(* IEC 61131-3 sources: plc_projects/St_Codes, 9 files *)

(* ---- GVL.st ---- *)
(* ==========================================
   POU: GVL
   ========================================== *)

=== DECLARATION ===
{attribute 'qualified_only'}
VAR_GLOBAL
    Recipe_Weights AT %MD100 : ARRAY[1..20] OF REAL;
	Auto_Bin_Material_Mapping AT %MW50: ARRAY[1..6] OF INT;
	Semi_Auto_Bin_Material_Mapping AT %MW60: ARRAY[1..10] OF INT;
	Auto_Coarse_To_Fine_speed AT %MD120: ARRAY[1..6] OF REAL := [1.0,1.0,1.0,1.0,1.0,1.0];
	Semi_Auto_Coarse_To_Fine_speed AT %MD130: ARRAY[1..10] OF REAL := [1.0,1.0,1.0,1.0,1.0,1.0,1.0,1.0,1.0,1.0];
	Auto_Bin_Tolerance AT %MD150: ARRAY[1..6] OF REAL;
	Semi_Auto_Bin_Tolerance AT %MD160: ARRAY[1..10] OF REAL;
	Start_Button AT %MX2.0: BOOL;
	E_Stop_Active AT %MX2.1: BOOL;
	Reset AT %MX2.3: BOOL;
	Next_Cycle_Start AT %MX2.4: BOOL;               // Command pulse/signal to start next batch cycle after hoppers are emptied
	Auto_Active_Mat AT %MW70: INT;
	Auto_Active_Bin AT %MW71: INT;
	Semi_Auto_Active_Mat AT %MW72: INT;
	Semi_Auto_Active_Bin AT %MW73: INT;
	Target_Batch_Cycles AT %MW74: INT := 1;
	Current_Batch_Cycle AT %MW75: INT;
	Completed_Batch_Cycles AT %MW79: INT;
	Error_Code AT %MW76: INT;
	Run AT %MX2.5 : BOOL;
	load_cell_auto AT %MD174 : REAL;
	load_cell_semi_auto AT %MD175 : REAL;
	Auto_Initial_Tolerance AT %MD176 : REAL := 5.0;
	Semi_Auto_Initial_Tolerance AT %MD178 : REAL := 5.0;
	Empty_Weight_Limit AT %MD186 : REAL := 5.0;     // Maximum scale weight limit (kg) to qualify scale as empty before starting next cycle
	Auto_Total_Target_Weight AT %MD180 : REAL;
	Semi_Auto_Total_Target_Weight AT %MD184 : REAL;
	Auto_Material_Count AT %MW77 : INT;
	Semi_Auto_Material_Count AT %MW78 : INT;
	Auto_Current_Step AT %MW80 : INT;
	Semi_Auto_Current_Step AT %MW81 : INT;
	Auto_Active_Target_Weight AT %MD220 : REAL;
	Semi_Auto_Active_Target_Weight AT %MD224 : REAL;
	Auto_Active_Live_Weight AT %MD228 : REAL;
	Semi_Auto_Active_Live_Weight AT %MD232 : REAL;
	Auto_Excess_Allowed AT %MX2.6 : BOOL;
	Semi_Auto_Excess_Allowed AT %MX2.9 : BOOL;
	Auto_Excess_Alarm AT %MX2.7 : BOOL;
	Semi_Auto_Excess_Alarm AT %MX2.8 : BOOL;
	Auto_Inter_Bin_Delay AT %MD190 : TIME;
	Semi_Auto_Inter_Bin_Delay AT %MD194 : TIME;
	Auto_Sequence_Complete AT %MX3.0 : BOOL;
	Semi_Auto_Sequence_Complete AT %MX3.1 : BOOL;
	All_Cycles_Complete AT %MX3.2 : BOOL;           // Master flag: TRUE when all target batch cycles have completed
	Auto_Status_Message : STRING(80);
	Semi_Auto_Status_Message : STRING(80);

	(* 8 Process Output and Weight Arrays *)
	Auto_Bin : ARRAY[1..6] OF BOOL;
	auto_bin_cutoff : ARRAY[1..6] OF BOOL;
	auto_bin_motor : ARRAY[1..6] OF BOOL;
	Semi_Auto_Bin : ARRAY[1..10] OF BOOL;
	semi_auto_bin_cutoff : ARRAY[1..10] OF BOOL;
	semi_auto_bin_motor : ARRAY[1..10] OF BOOL;
	Auto_Weights : ARRAY[1..6] OF REAL;
	Semi_Auto_Weights : ARRAY[1..10] OF REAL;
END_VAR

(* ---- Auto_Batching_V13.st ---- *)
FUNCTION_BLOCK Auto_Batching_V13
VAR_INPUT
    Start_Button : BOOL;      // Signal to start/resume the batching sequence
    E_Stop_Active : BOOL;     // Emergency Stop (Pause/Hold signal)
    Reset : BOOL;             // Hard reset sequence trigger
    Auto_Bin_Material_Mapping : ARRAY[1..6] OF INT; // Material index mapping for 6 bins
    Auto_Coarse_To_Fine_speed : ARRAY[1..6] OF REAL; // Cutoff weight thresholds (kg)
    Auto_Bin_Tolerance : ARRAY[1..6] OF REAL; // Tolerance weight offset values (kg)
    Inter_Bin_Delay : TIME;   // Global inter-bin delay time
    Excess_Allowed : BOOL;    // Global toggle: TRUE = skip excess check, FALSE = trigger alarm & hold
END_VAR
VAR_IN_OUT
    load_cell_value : REAL;   // Weight value read/written from load cell
END_VAR
VAR_OUTPUT
    Auto_Bin : ARRAY[1..6] OF BOOL; // Coarse feed valve outputs
    auto_bin_cutoff : ARRAY[1..6] OF BOOL; // Fine feed cutoff trigger indicators
    auto_bin_motor : ARRAY[1..6] OF BOOL; // Main conveyor motor outputs
    Actual_Weights : ARRAY[1..6] OF REAL; // Actual weight poured per silo
    Sequence_Complete : BOOL;  // Batch complete flag
    Active_Material_ID : INT;  // Currently active ingredient ID
    Active_Bin_ID : INT;       // Currently active physical Bin ID (1..6)
    Active_Target_Weight : REAL; // Recipe target weight of active bin
    Active_Live_Weight : REAL; // Live tared weight poured from active bin
    Excess_Alarm : BOOL;       // Excess weight alarm output
    Error_Code : INT;          // Active error code
    Status_Message : STRING;   // Diagnostic text message
END_VAR
VAR
    Step : INT;                // State machine index (0: Idle, 1..6: Pour, 7: Settling, 8: Complete)
    bin_last_weight : REAL;   // Baseline weight snapshot before starting current bin
    actual_bin : REAL;        // Current weight added from active bin
    target_weight : REAL;     // Target recipe weight
    cutoff_trigger_weight : REAL; // Calculated cutoff trigger threshold (Target - Cutoff)
    min_tol_weight : REAL;    // Minimum allowable tolerance (Target - Tol)
    max_tol_weight : REAL;    // Maximum allowable tolerance (Target + Tol)
    Paused_By_EStop : BOOL;    // Pause status latch
    Effective_Delay : TIME;   // Resolved delay time (defaults to T#2S if T#0S configured)

    Mat_Idx : INT;
    i : INT;                  // General loop index

    (* TIMERS FOR TRANSITIONS & DELAYS *)
    Transition_Timer : TON;
    Completion_Timer : TON;

    (* SELF-CONTAINED SIMULATION VARIABLES *)
    Simulation_Mode : BOOL;    // Simulation disabled for physical PLC use
    Sim_Rate : REAL;
    Sim_Timer : TON;
    Start_Sim_Weight : REAL;
    Discharge_Active : BOOL;
END_VAR

(* Auto Batching FB V13 with Real-Time Instant Excess Verification & Clean Multi-Cycle Reset *)

Effective_Delay := Inter_Bin_Delay;
IF Effective_Delay = T#0S THEN
    Effective_Delay := T#2S;
END_IF;

(* 1. HARD RESET INTERLOCK *)
IF Reset THEN
    FOR i := 1 TO 6 DO
        Auto_Bin[i] := FALSE;
        auto_bin_cutoff[i] := FALSE;
        auto_bin_motor[i] := FALSE;
        Actual_Weights[i] := 0.0;
    END_FOR;
    Sequence_Complete := FALSE;
    Active_Material_ID := 0;
    Active_Bin_ID := 0;
    Active_Target_Weight := 0.0;
    Active_Live_Weight := 0.0;
    Excess_Alarm := FALSE;
    Error_Code := 0;
    Status_Message := '';
    Paused_By_EStop := FALSE;
    Step := 0;

    bin_last_weight := 0.0;
    Start_Sim_Weight := 0.0;

    Transition_Timer(IN := FALSE);
    Completion_Timer(IN := FALSE);
    Sim_Timer(IN := FALSE);
    RETURN;
END_IF;

(* 2. E-STOP PAUSE / HOLD LOGIC *)
IF E_Stop_Active THEN
    Paused_By_EStop := TRUE;
END_IF;

IF Paused_By_EStop THEN
    FOR i := 1 TO 6 DO
        Auto_Bin[i] := FALSE;
        auto_bin_cutoff[i] := FALSE;
        auto_bin_motor[i] := FALSE;
    END_FOR;

    IF E_Stop_Active THEN
        Status_Message := 'Auto Paused: Emergency Stop Active!';
    ELSE
        Status_Message := 'Auto Paused: Press Start to Resume';
        IF Start_Button THEN
            Paused_By_EStop := FALSE;
        END_IF;
    END_IF;

    Sim_Timer(IN := FALSE);
    Transition_Timer(IN := FALSE);
    Completion_Timer(IN := FALSE);
    RETURN;
END_IF;

(* 3. SIMULATION WEIGHT MANAGEMENT (WHEN ENABLED) *)
IF Simulation_Mode THEN
    IF Step = 0 AND NOT Start_Button AND NOT Sequence_Complete THEN
        load_cell_value := 0.0;
        bin_last_weight := 0.0;
        Start_Sim_Weight := 0.0;
        Sim_Timer(IN := FALSE);
    END_IF;

    Discharge_Active := FALSE;
    IF Step >= 1 AND Step <= 6 THEN
        Discharge_Active := auto_bin_motor[Step];
    END_IF;

    IF Discharge_Active THEN
        Sim_Timer(IN := TRUE, PT := T#1000S);
        load_cell_value := Start_Sim_Weight + (TIME_TO_REAL(Sim_Timer.ET) / 1000.0) * Sim_Rate;
    ELSE
        Sim_Timer(IN := FALSE);
        Start_Sim_Weight := load_cell_value;
    END_IF;
END_IF;

(* 4. RECIPE SEQUENCE START & CYCLIC RESET *)
IF Step = 0 AND Start_Button THEN
    Step := 1;
    bin_last_weight := load_cell_value; (* Snapshot relative tare at whatever weight scale is *)
    Sequence_Complete := FALSE;
    Excess_Alarm := FALSE;
    Error_Code := 0;
    Status_Message := 'Auto Pour Started';
    Active_Target_Weight := 0.0;
    Active_Live_Weight := 0.0;
    FOR i := 1 TO 6 DO
        Actual_Weights[i] := 0.0;
        Auto_Bin[i] := FALSE;
        auto_bin_cutoff[i] := FALSE;
        auto_bin_motor[i] := FALSE;
    END_FOR;
END_IF;

(* 5. SEQUENCE CONTROL STATE MACHINE *)
CASE Step OF
    0:
        Active_Material_ID := 0;
        Active_Bin_ID := 0;
        Active_Target_Weight := 0.0;
        Active_Live_Weight := 0.0;
        Excess_Alarm := FALSE;
        Sequence_Complete := FALSE;
        FOR i := 1 TO 6 DO
            Auto_Bin[i] := FALSE;
            auto_bin_cutoff[i] := FALSE;
            auto_bin_motor[i] := FALSE;
        END_FOR;
        IF Error_Code = 0 THEN Status_Message := 'Auto Idle'; END_IF;

    1..6: (* DISCHARGE SILOS 1 TO 6 *)
        Mat_Idx := Auto_Bin_Material_Mapping[Step];

        (* Skip this step instantly if material mapping is 0 OR target weight is 0.0 kg *)
        IF Mat_Idx = 0 OR (Mat_Idx <= 20 AND GVL.Recipe_Weights[Mat_Idx] = 0.0) THEN
            IF Step = 6 THEN
                Step := 7; (* Transition directly to final settling delay *)
            ELSE
                Step := Step + 1;
            END_IF;
        ELSE
            target_weight := GVL.Recipe_Weights[Mat_Idx];
            cutoff_trigger_weight := target_weight - Auto_Coarse_To_Fine_speed[Step];
            min_tol_weight := target_weight - Auto_Bin_Tolerance[Step];
            max_tol_weight := target_weight + Auto_Bin_Tolerance[Step];

            Active_Target_Weight := target_weight;
            actual_bin := load_cell_value - bin_last_weight;
            Actual_Weights[Step] := actual_bin;
            Active_Live_Weight := actual_bin; (* Live tared weight of active bin *)

            Active_Material_ID := Mat_Idx;
            Active_Bin_ID := Step;

            (* Scale Overload Protection *)
            IF load_cell_value > 500.0 THEN
                Error_Code := 21;
                Status_Message := 'Error 21: Scale Overloaded!';
                Sequence_Complete := TRUE;
                Paused_By_EStop := TRUE;
            END_IF;

            (* Real-Time Feed & Instant Excess Alarm *)
            IF actual_bin < cutoff_trigger_weight THEN
                (* Coarse Feed *)
                Auto_Bin[Step] := TRUE;
                auto_bin_cutoff[Step] := FALSE;
                auto_bin_motor[Step] := TRUE;
                Excess_Alarm := FALSE;
                Status_Message := 'Auto Pouring (Coarse Feed)';

            ELSIF actual_bin < min_tol_weight THEN
                (* Fine Feed *)
                Auto_Bin[Step] := FALSE;
                auto_bin_cutoff[Step] := TRUE;
                auto_bin_motor[Step] := TRUE;
                Excess_Alarm := FALSE;
                Status_Message := 'Auto Pouring (Fine Feed)';

            ELSIF actual_bin > max_tol_weight THEN
                (* Excess Weight -> Instant Alarm, No Delay! *)
                Auto_Bin[Step] := FALSE;
                auto_bin_cutoff[Step] := FALSE;
                auto_bin_motor[Step] := FALSE;

                IF Excess_Allowed THEN
                    Excess_Alarm := FALSE;
                    Status_Message := 'Excess Weight Allowed: Advancing';
                    bin_last_weight := load_cell_value;
                    Active_Target_Weight := 0.0;
                    Active_Live_Weight := 0.0;
                    IF Step = 6 THEN
                        Step := 7;
                    ELSE
                        Step := Step + 1;
                    END_IF;
                ELSE
                    Excess_Alarm := TRUE; (* Immediate Trigger! *)
                    Status_Message := 'Excess Alarm: Weight above max tolerance! Reduce weight.';
                END_IF;

            ELSE
                (* In Tolerance Window [Min_Tol .. Max_Tol] *)
                Auto_Bin[Step] := FALSE;
                auto_bin_cutoff[Step] := FALSE;
                auto_bin_motor[Step] := FALSE;
                Excess_Alarm := FALSE;
                bin_last_weight := load_cell_value;
                Active_Target_Weight := 0.0;
                Active_Live_Weight := 0.0;

                IF Step = 6 THEN
                    Step := 7;
                ELSE
                    Step := Step + 1;
                END_IF;
            END_IF;
        END_IF;

    7: (* POST-SEQUENCE FINAL SETTLING DELAY *)
        Active_Material_ID := 0;
        Active_Bin_ID := 0;
        Active_Target_Weight := 0.0;
        Active_Live_Weight := 0.0;
        Excess_Alarm := FALSE;
        Status_Message := 'Final Settling Delay';
        Completion_Timer(IN := TRUE, PT := Effective_Delay);
        IF Completion_Timer.Q THEN
            Completion_Timer(IN := FALSE);
            Step := 8;
        END_IF;

    8: (* COMPLETE *)
        Active_Material_ID := 0;
        Active_Bin_ID := 0;
        Active_Target_Weight := 0.0;
        Active_Live_Weight := 0.0;
        Excess_Alarm := FALSE;
        Status_Message := 'Sequence Completed';
        Sequence_Complete := TRUE;

        IF NOT Start_Button THEN
            Step := 0;
            Sequence_Complete := FALSE;
            FOR i := 1 TO 6 DO
                Actual_Weights[i] := 0.0;
            END_FOR;
        END_IF;
END_CASE;

(* ---- Auto_Batching_V14.st ---- *)
FUNCTION_BLOCK Auto_Batching_V14
VAR_INPUT
    Start_Button : BOOL;                            // Command pulse/signal to start or resume the auto batching sequence
    E_Stop_Active : BOOL;                           // Emergency Stop circuit status (NC contact: TRUE = Healthy/Run permitted, FALSE = E-Stop tripped)
    Reset : BOOL;                                   // System reset pulse (clears active steps, outputs, alarms, and error flags)
    Auto_Bin_Material_Mapping : ARRAY[1..6] OF INT; // Array mapping physical Silos 1..6 to Recipe Material IDs (1..20, 0 = Silo skipped)
    Auto_Coarse_To_Fine_Speed : ARRAY[1..6] OF REAL;// Weight offset threshold (kg) before target to transition from Coarse to Fine feeding
    Auto_Bin_Tolerance : ARRAY[1..6] OF REAL;       // Allowable weight tolerance window (±kg) around target weight for each silo
    Inter_Bin_Delay : TIME;                         // Settling delay duration after completing a bin before advancing to the next
    Excess_Allowed : BOOL;                          // Overfill handling policy: TRUE = proceed if target is exceeded, FALSE = raise alarm and halt
    load_cell_value : REAL;                         // Live gross weight input reading from the Auto scale load cell (kg)
    Target_Batch_Cycles : INT;                      // Target number of batch cycle repetitions configured from HMI (defaults to 1)
    Next_Cycle_Start : BOOL;                        // Command pulse/signal to start next batch cycle after hoppers are emptied
    Empty_Weight_Limit : REAL;                      // Maximum scale weight limit (kg) for scales to qualify as empty before starting next cycle
END_VAR
VAR_OUTPUT
    Auto_Bin : ARRAY[1..6] OF BOOL;                 // Coarse feeding valve / gate actuation command outputs for Silos 1..6
    auto_bin_cutoff : ARRAY[1..6] OF BOOL;          // Fine feeding valve / vibrator cutoff actuation command outputs for Silos 1..6
    auto_bin_motor : ARRAY[1..6] OF BOOL;           // Feeder / screw conveyor motor run commands for Silos 1..6
    Actual_Weights : ARRAY[1..6] OF REAL;           // Net material weight (kg) successfully dosed for each silo in the current cycle
    Sequence_Complete : BOOL;                       // Handshake flag: TRUE when all mapped Auto silos have completed dosing and settling
    Active_Material_ID : INT;                       // Recipe Material ID currently being dosed (1..20, 0 when idle/complete)
    Active_Bin_ID : INT;                            // Physical Silo index currently being dosed (1..6, 0 when idle/complete)
    Active_Target_Weight : REAL;                    // Target weight setpoint (kg) of the ingredient currently being dosed
    Active_Live_Weight : REAL;                      // Live net/tared weight (kg) accumulated into the scale for the active silo
    Current_Step : INT;                             // Real-time sequence step:
                                                    //   0  = Idle / Waiting for Start
                                                    //   1..6 = Dosing Silos 1..6 (feeding coarse/fine)
                                                    //   7  = Settling delay in progress
                                                    //   8  = Sequence complete
    Cycle_Manager_State : INT;                      // Master supervisory cycle manager state:
                                                    //   0  = System Idle / Stopped
                                                    //   1  = Running active batch cycle
                                                    //   4  = All target batch cycles completed successfully
                                                    //   5  = Paused between cycles (Cycle Hold active)
    Excess_Alarm : BOOL;                            // Overfill alarm: TRUE when dosed weight exceeds target + tolerance (with Excess_Allowed=FALSE)
    Error_Code : INT;                               // Fault diagnostic code:
                                                    //   0  = No Error / System Healthy
                                                    //   1  = Duplicate Material ID mapped across Auto and Semi-Auto
                                                    //   2  = Material index out of range (must be 1..20)
                                                    //   3  = Recipe weight is less than (Coarse_To_Fine_Speed + Tolerance)
                                                    //   4  = Initial scale tare error (scale not empty before start)
                                                    //   21 = Scale overload protection triggered (> 500 kg)
    Auto_Current_Batch_Cycle : INT;                     // Active batch cycle number currently processing (1..Target_Batch_Cycles)
    Auto_Completed_Batch_Cycles : INT;                  // Total number of batch cycle loops completed successfully
    Auto_All_Cycles_Complete : BOOL;                    // Master flag: TRUE when all Target_Batch_Cycles have finished
    Status_Message : STRING(80);                    // Real-time human-readable process status and diagnostic text message
END_VAR
VAR
    bin_last_weight : REAL;
    actual_bin : REAL;
    target_weight : REAL;
    cutoff_trigger_weight : REAL;
    min_tol_weight : REAL;
    max_tol_weight : REAL;
    Paused_By_EStop : BOOL;
    Effective_Delay : TIME;
    Mat_Idx : INT;
    i : INT;
    j : INT;
    Transition_Timer : TON;
    Completion_Timer : TON;
    Simulation_Mode : BOOL;
    Sim_Rate : REAL;
    Sim_Timer : TON;
    Start_Sim_Weight : REAL;
    Discharge_Active : BOOL;

    (* Master Cycle Manager & Supervisory states *)
    Internal_FB_Start : BOOL;
    Duplicate_Found : BOOL;
    Invalid_Material_Range : BOOL;
    Weight_Limit_Error : BOOL;
    eff_empty_limit : REAL;
    Next_Cycle_Last : BOOL;
    Next_Cycle_Rising : BOOL;
END_VAR

(* Auto Batching FB V14 with Full Diagnostics, Step Tracking, and Precise Status Reporting *)

Effective_Delay := Inter_Bin_Delay;
IF Effective_Delay = T#0S THEN
    Effective_Delay := T#2S;
END_IF;

(* Detect rising edge on Next_Cycle_Start trigger *)
Next_Cycle_Rising := (Next_Cycle_Start OR GVL.Next_Cycle_Start) AND NOT Next_Cycle_Last;
Next_Cycle_Last := (Next_Cycle_Start OR GVL.Next_Cycle_Start);

(* 1. RECIPE TOTALS & SUPERVISORY CONFIGURATION CHECKS *)
Duplicate_Found := FALSE;
Invalid_Material_Range := FALSE;
Weight_Limit_Error := FALSE;

GVL.Auto_Total_Target_Weight := 0.0;
GVL.Auto_Material_Count := 0;
FOR i := 1 TO 6 DO
    IF Auto_Bin_Material_Mapping[i] < 0 OR Auto_Bin_Material_Mapping[i] > 20 THEN
        Invalid_Material_Range := TRUE;
    END_IF;
    IF Auto_Bin_Material_Mapping[i] <> 0 AND Auto_Bin_Material_Mapping[i] <= 20 THEN
        FOR j := 1 TO 10 DO
            IF Auto_Bin_Material_Mapping[i] = GVL.Semi_Auto_Bin_Material_Mapping[j] THEN
                Duplicate_Found := TRUE;
            END_IF;
        END_FOR;
    END_IF;
    IF Auto_Bin_Material_Mapping[i] > 0 AND Auto_Bin_Material_Mapping[i] <= 20 THEN
        IF GVL.Recipe_Weights[Auto_Bin_Material_Mapping[i]] > 0.0 THEN
            GVL.Auto_Total_Target_Weight := GVL.Auto_Total_Target_Weight + GVL.Recipe_Weights[Auto_Bin_Material_Mapping[i]];
            GVL.Auto_Material_Count := GVL.Auto_Material_Count + 1;
            IF GVL.Recipe_Weights[Auto_Bin_Material_Mapping[i]] < (Auto_Coarse_To_Fine_Speed[i] + Auto_Bin_Tolerance[i]) THEN
                Weight_Limit_Error := TRUE;
            END_IF;
        END_IF;
    END_IF;
END_FOR;

IF Duplicate_Found THEN
    GVL.Error_Code := 1;
    Error_Code := 1;
    Status_Message := 'Error 1: Duplicate Material ID mapped in Auto and Semi-Auto!';
ELSIF Invalid_Material_Range THEN
    GVL.Error_Code := 2;
    Error_Code := 2;
    Status_Message := 'Error 2: Material Index configuration out of range (1..20)!';
ELSIF Weight_Limit_Error THEN
    GVL.Error_Code := 3;
    Error_Code := 3;
    Status_Message := 'Error 3: Recipe weight is less than Coarse_To_Fine_Speed + Tolerance!';
ELSE
    IF GVL.Error_Code <= 3 THEN
        GVL.Error_Code := 0;
        Error_Code := 0;
    END_IF;
END_IF;

(* 2. HARD RESET INTERLOCK *)
IF Reset OR GVL.Reset THEN
    FOR i := 1 TO 6 DO
        Auto_Bin[i] := FALSE;
        auto_bin_cutoff[i] := FALSE;
        auto_bin_motor[i] := FALSE;
        Actual_Weights[i] := 0.0;
        GVL.Auto_Bin[i] := FALSE;
        GVL.auto_bin_cutoff[i] := FALSE;
        GVL.auto_bin_motor[i] := FALSE;
        GVL.Auto_Weights[i] := 0.0;
    END_FOR;

    (* Reset Recipe & Active Target Setpoints *)
    FOR i := 1 TO 20 DO
        GVL.Recipe_Weights[i] := 0.0;
    END_FOR;
    GVL.Auto_Total_Target_Weight := 0.0;
    GVL.Semi_Auto_Total_Target_Weight := 0.0;
    GVL.Auto_Material_Count := 0;
    GVL.Semi_Auto_Material_Count := 0;

    Sequence_Complete := FALSE;
    GVL.Auto_Sequence_Complete := FALSE;
    GVL.Semi_Auto_Sequence_Complete := FALSE;
    Active_Material_ID := 0;
    Active_Bin_ID := 0;
    Active_Target_Weight := 0.0;
    Active_Live_Weight := 0.0;
    GVL.Auto_Active_Target_Weight := 0.0;
    GVL.Auto_Active_Live_Weight := 0.0;
    Excess_Alarm := FALSE;
    Error_Code := 0;
    GVL.Error_Code := 0;
    GVL.Current_Batch_Cycle := 0;
    GVL.Completed_Batch_Cycles := 0;
    GVL.All_Cycles_Complete := FALSE;
    Auto_Completed_Batch_Cycles := 0;
    Auto_Current_Batch_Cycle := 0;
    Auto_All_Cycles_Complete := FALSE;
    GVL.Target_Batch_Cycles := 0;
    GVL.Start_Button := FALSE;
    GVL.Run := FALSE;
    GVL.Next_Cycle_Start := FALSE;
    Next_Cycle_Last := FALSE;
    Next_Cycle_Rising := FALSE;
    GVL.Auto_Active_Mat := 0;
    GVL.Auto_Active_Bin := 0;
    GVL.Auto_Excess_Alarm := FALSE;
    Current_Step := 0;
    Cycle_Manager_State := 0;
    Internal_FB_Start := FALSE;
    bin_last_weight := 0.0;
    Start_Sim_Weight := 0.0;
    Transition_Timer(IN := FALSE);
    Completion_Timer(IN := FALSE);
    Sim_Timer(IN := FALSE);
    Status_Message := 'Auto [Reset]: System Reset Complete - System Idle';
    RETURN;
END_IF;

(* 3. E-STOP PAUSE / HOLD LOGIC (NC Contact: FALSE = Pressed/Tripped, TRUE = Healthy) *)
IF NOT E_Stop_Active OR NOT GVL.E_Stop_Active THEN
    Paused_By_EStop := TRUE;
END_IF;

IF Paused_By_EStop THEN
    FOR i := 1 TO 6 DO
        Auto_Bin[i] := FALSE;
        auto_bin_cutoff[i] := FALSE;
        auto_bin_motor[i] := FALSE;
    END_FOR;
    IF NOT E_Stop_Active OR NOT GVL.E_Stop_Active THEN
        Status_Message := CONCAT('Auto [PAUSED]: E-Stop Active at Step ', INT_TO_STRING(Current_Step));
    ELSE
        Status_Message := CONCAT('Auto [HOLD]: E-Stop Cleared. Press Start to Resume Step ', INT_TO_STRING(Current_Step));
        IF Start_Button OR GVL.Start_Button THEN
            Paused_By_EStop := FALSE;
        END_IF;
    END_IF;
    Sim_Timer(IN := FALSE);
    Transition_Timer(IN := FALSE);
    Completion_Timer(IN := FALSE);
    RETURN;
END_IF;

(* 4. MASTER CYCLE MANAGER STATE MACHINE *)
CASE Cycle_Manager_State OF
    0: (* IDLE *)
        Internal_FB_Start := FALSE;
        GVL.Run := FALSE;
        GVL.Next_Cycle_Start := FALSE;
        GVL.Auto_Sequence_Complete := FALSE;

        IF GVL.Error_Code = 0 AND NOT (Start_Button OR GVL.Start_Button) THEN
            Status_Message := 'Auto [State 0 - Idle]: Ready - Waiting for Start Button';
        END_IF;

        IF Start_Button OR GVL.Start_Button THEN
            (* Use Target_Batch_Cycles from input, or fallback to GVL, or default to 1 *)
            IF Target_Batch_Cycles > 0 THEN
                GVL.Target_Batch_Cycles := Target_Batch_Cycles;
            ELSIF GVL.Target_Batch_Cycles <= 0 THEN
                GVL.Target_Batch_Cycles := 1;
            END_IF;

            IF NOT E_Stop_Active OR NOT GVL.E_Stop_Active THEN
                GVL.Run := FALSE;
                Status_Message := 'Auto [State 0]: Cannot Start - Emergency Stop Contact Open!';
            ELSIF (GVL.Auto_Initial_Tolerance > 0.0 AND (GVL.load_cell_auto > GVL.Auto_Initial_Tolerance OR GVL.load_cell_auto < (-GVL.Auto_Initial_Tolerance))) OR
                  (GVL.Semi_Auto_Initial_Tolerance > 0.0 AND (GVL.load_cell_semi_auto > GVL.Semi_Auto_Initial_Tolerance OR GVL.load_cell_semi_auto < (-GVL.Semi_Auto_Initial_Tolerance))) THEN
                GVL.Run := FALSE;
                GVL.Error_Code := 4;
                Error_Code := 4;
                Status_Message := 'Auto [State 0]: Error 4 - Scale not zeroed (exceeds Initial Tolerance)!';
            ELSE
                GVL.Error_Code := 0;
                Error_Code := 0;
                GVL.Current_Batch_Cycle := 1;
                GVL.Completed_Batch_Cycles := 0;
                GVL.All_Cycles_Complete := FALSE;
                Auto_Completed_Batch_Cycles := 0;
                Auto_Current_Batch_Cycle := 1;
                Auto_All_Cycles_Complete := FALSE;
                GVL.Run := TRUE;
                Internal_FB_Start := TRUE;
                Sequence_Complete := FALSE;
                GVL.Auto_Sequence_Complete := FALSE;
                GVL.Semi_Auto_Sequence_Complete := FALSE;
                Cycle_Manager_State := 1;
                Current_Step := 0;
            END_IF;
        END_IF;

    1: (* RUNNING CYCLE *)
        Internal_FB_Start := TRUE;
        GVL.Run := TRUE;

        (* Interlock: While process is actively running, Next_Cycle_Start MUST be FALSE *)
        GVL.Next_Cycle_Start := FALSE;

        (* Both Auto and Semi-Auto must complete to finish the cycle *)
        IF Sequence_Complete AND GVL.Semi_Auto_Sequence_Complete THEN
            GVL.Completed_Batch_Cycles := GVL.Current_Batch_Cycle;
            Auto_Completed_Batch_Cycles := GVL.Current_Batch_Cycle;
            IF GVL.Current_Batch_Cycle < GVL.Target_Batch_Cycles AND GVL.Error_Code = 0 THEN
                Internal_FB_Start := FALSE;
                Cycle_Manager_State := 5; (* Go to pause/hold to wait for scale empty & Next_Cycle_Start *)
            ELSE
                Cycle_Manager_State := 4; (* All target cycles completed *)
            END_IF;
        END_IF;

    5: (* PAUSED BETWEEN CYCLES - WAITING FOR HOPPERS EMPTIED & NEXT CYCLE START *)
        Internal_FB_Start := FALSE;
        GVL.Run := TRUE;

        (* Determine effective empty weight threshold (defaults to 5.0 kg if <= 0.0) *)
        eff_empty_limit := Empty_Weight_Limit;
        IF eff_empty_limit <= 0.0 THEN
            eff_empty_limit := GVL.Empty_Weight_Limit;
        END_IF;
        IF eff_empty_limit <= 0.0 THEN
            eff_empty_limit := 5.0;
        END_IF;

        Status_Message := CONCAT('Auto [State 5]: Cycle ', CONCAT(INT_TO_STRING(GVL.Current_Batch_Cycle), ' Done. Empty scales < limit and trigger Next_Cycle_Start.'));

        (* Check ONLY on a new trigger pulse (rising edge) of Next_Cycle_Start *)
        IF Next_Cycle_Rising THEN
            (* Check both scales are below the empty weight limit at the moment of trigger *)
            IF (GVL.load_cell_auto < eff_empty_limit) AND (GVL.load_cell_semi_auto < eff_empty_limit) THEN
                (* Scale is empty: momentary reset of command, advance to next cycle *)
                GVL.Next_Cycle_Start := FALSE;
                Next_Cycle_Last := FALSE;
                GVL.Start_Button := TRUE; (* Keep Start_Button TRUE until all cycles are complete! *)
                GVL.Error_Code := 0;
                Error_Code := 0;
                GVL.Current_Batch_Cycle := GVL.Current_Batch_Cycle + 1;
                Auto_Current_Batch_Cycle := GVL.Current_Batch_Cycle;
                Sequence_Complete := FALSE;
                GVL.Auto_Sequence_Complete := FALSE;
                GVL.Semi_Auto_Sequence_Complete := FALSE;
                Current_Step := 0;
                Internal_FB_Start := TRUE;
                Cycle_Manager_State := 1;
                FOR i := 1 TO 6 DO
                    Actual_Weights[i] := 0.0;
                    Auto_Bin[i] := FALSE;
                    auto_bin_cutoff[i] := FALSE;
                    auto_bin_motor[i] := FALSE;
                END_FOR;
            ELSE
                (* Scale not empty yet: reject trigger, reset command, and wait for operator to trigger again *)
                GVL.Next_Cycle_Start := FALSE;
                Next_Cycle_Last := FALSE;
                Status_Message := CONCAT('Auto [State 5]: Scale weight exceeds limit (', CONCAT(REAL_TO_STRING(eff_empty_limit), ' kg)! Empty scales and trigger Next_Cycle_Start again.'));
            END_IF;
        END_IF;

    4: (* ALL CYCLES COMPLETE *)
        Internal_FB_Start := FALSE;
        GVL.Run := FALSE;
        GVL.Start_Button := FALSE;
        Auto_All_Cycles_Complete := TRUE;
        GVL.All_Cycles_Complete := TRUE;
        Sequence_Complete := TRUE;
        GVL.Auto_Sequence_Complete := TRUE;
        GVL.Semi_Auto_Sequence_Complete := TRUE;
        Status_Message := CONCAT('Auto [State 4 - Finished]: All ', CONCAT(INT_TO_STRING(GVL.Target_Batch_Cycles), ' Batch Cycles Completed Successfully'));
        IF Start_Button OR GVL.Start_Button THEN
            (* Reset flags for new batch start *)
            Current_Step := 0;
            Auto_All_Cycles_Complete := FALSE;
            GVL.All_Cycles_Complete := FALSE;
            Sequence_Complete := FALSE;
            GVL.Auto_Sequence_Complete := FALSE;
            GVL.Semi_Auto_Sequence_Complete := FALSE;
            Cycle_Manager_State := 0;
        END_IF;
END_CASE;

(* 5. AUTO SILOS 1..6 POURING SEQUENCE WITH DETAILED STATUS *)
IF Current_Step = 0 AND Internal_FB_Start THEN
    Current_Step := 1;
    bin_last_weight := load_cell_value;
    Sequence_Complete := FALSE;
    GVL.Auto_Sequence_Complete := FALSE;
    Excess_Alarm := FALSE;
    Error_Code := 0;
    FOR i := 1 TO 6 DO
        Actual_Weights[i] := 0.0;
        Auto_Bin[i] := FALSE;
        auto_bin_cutoff[i] := FALSE;
        auto_bin_motor[i] := FALSE;
    END_FOR;
END_IF;

CASE Current_Step OF
    0:
        Active_Material_ID := 0;
        Active_Bin_ID := 0;
        Excess_Alarm := FALSE;
        Sequence_Complete := FALSE;
        FOR i := 1 TO 6 DO
            Auto_Bin[i] := FALSE;
            auto_bin_cutoff[i] := FALSE;
            auto_bin_motor[i] := FALSE;
        END_FOR;
        Active_Target_Weight := GVL.Auto_Active_Target_Weight;
        Active_Live_Weight := 0.0;

    1..6:
        (* Skip any bin where Material Mapping is 0, > 20, or Recipe Weight is 0 *)
        WHILE Current_Step >= 1 AND Current_Step <= 6 DO
            Mat_Idx := Auto_Bin_Material_Mapping[Current_Step];
            IF Mat_Idx = 0 OR Mat_Idx > 20 OR GVL.Recipe_Weights[Mat_Idx] <= 0.0 THEN
                Auto_Bin[Current_Step] := FALSE;
                auto_bin_cutoff[Current_Step] := FALSE;
                auto_bin_motor[Current_Step] := FALSE;
                Actual_Weights[Current_Step] := 0.0;
                IF Current_Step = 6 THEN
                    Current_Step := 7;
                    EXIT;
                ELSE
                    Current_Step := Current_Step + 1;
                END_IF;
            ELSE
                EXIT; (* Valid active recipe silo found *)
            END_IF;
        END_WHILE;

        IF Current_Step = 7 THEN
            Active_Material_ID := 0;
            Active_Bin_ID := 0;
            Active_Target_Weight := 0.0;
            Active_Live_Weight := 0.0;
            GVL.Auto_Active_Target_Weight := 0.0;
            GVL.Auto_Active_Live_Weight := 0.0;
            Status_Message := 'Auto [Step 7]: Settling Delay in progress...';
            Completion_Timer(IN := TRUE, PT := Effective_Delay);
            IF Completion_Timer.Q THEN
                Completion_Timer(IN := FALSE);
                Current_Step := 8;
            END_IF;
        ELSE
            Mat_Idx := Auto_Bin_Material_Mapping[Current_Step];
            target_weight := GVL.Recipe_Weights[Mat_Idx];

            Active_Target_Weight := target_weight;
            GVL.Auto_Active_Target_Weight := target_weight;

            cutoff_trigger_weight := target_weight - Auto_Coarse_To_Fine_Speed[Current_Step];
            min_tol_weight := target_weight - Auto_Bin_Tolerance[Current_Step];
            max_tol_weight := target_weight + Auto_Bin_Tolerance[Current_Step];

            actual_bin := load_cell_value - bin_last_weight;
            IF actual_bin < 0.0 THEN
                actual_bin := 0.0;
            END_IF;
            Actual_Weights[Current_Step] := actual_bin;
            Active_Live_Weight := actual_bin;
            GVL.Auto_Active_Live_Weight := actual_bin;
            Active_Material_ID := Mat_Idx;
            Active_Bin_ID := Current_Step;

            IF load_cell_value > 500.0 THEN
                Error_Code := 21;
                GVL.Error_Code := 21;
                Status_Message := CONCAT('Auto [Step ', CONCAT(INT_TO_STRING(Current_Step), ']: STUCK - Error 21: Scale Overloaded (> 500 kg)!'));
                Sequence_Complete := TRUE;
                GVL.Auto_Sequence_Complete := TRUE;
                Paused_By_EStop := TRUE;
            END_IF;

            IF actual_bin < cutoff_trigger_weight THEN
                Auto_Bin[Current_Step] := TRUE;
                auto_bin_cutoff[Current_Step] := FALSE;
                auto_bin_motor[Current_Step] := TRUE;
                Excess_Alarm := FALSE;
                Status_Message := CONCAT('Auto [Step ', CONCAT(INT_TO_STRING(Current_Step), ']: Coarse Feeding'));
            ELSIF actual_bin < min_tol_weight THEN
                Auto_Bin[Current_Step] := FALSE;
                auto_bin_cutoff[Current_Step] := TRUE;
                auto_bin_motor[Current_Step] := TRUE;
                Excess_Alarm := FALSE;
                Status_Message := CONCAT('Auto [Step ', CONCAT(INT_TO_STRING(Current_Step), ']: Fine Feeding'));
            ELSIF actual_bin > max_tol_weight THEN
                Auto_Bin[Current_Step] := FALSE;
                auto_bin_cutoff[Current_Step] := FALSE;
                auto_bin_motor[Current_Step] := FALSE;
                IF Excess_Allowed THEN
                    Excess_Alarm := FALSE;
                    Status_Message := CONCAT('Auto [Step ', CONCAT(INT_TO_STRING(Current_Step), ']: Excess Allowed - Advancing'));
                    bin_last_weight := load_cell_value;
                    Active_Target_Weight := 0.0;
                    Active_Live_Weight := 0.0;
                    GVL.Auto_Active_Target_Weight := 0.0;
                    GVL.Auto_Active_Live_Weight := 0.0;
                    IF Current_Step = 6 THEN
                        Current_Step := 7;
                    ELSE
                        Current_Step := Current_Step + 1;
                    END_IF;
                ELSE
                    Excess_Alarm := TRUE;
                    Status_Message := CONCAT('Auto [Step ', CONCAT(INT_TO_STRING(Current_Step), ']: STUCK - Excess Weight! Reduce weight or enable Excess Allowed.'));
                END_IF;
            ELSE
                Auto_Bin[Current_Step] := FALSE;
                auto_bin_cutoff[Current_Step] := FALSE;
                auto_bin_motor[Current_Step] := FALSE;
                Excess_Alarm := FALSE;
                bin_last_weight := load_cell_value;
                Active_Target_Weight := 0.0;
                Active_Live_Weight := 0.0;
                GVL.Auto_Active_Target_Weight := 0.0;
                GVL.Auto_Active_Live_Weight := 0.0;
                Status_Message := CONCAT('Auto [Step ', CONCAT(INT_TO_STRING(Current_Step), ']: Target Reached - Advancing'));
                IF Current_Step = 6 THEN
                    Current_Step := 7;
                ELSE
                    Current_Step := Current_Step + 1;
                END_IF;
            END_IF;
        END_IF;

    7:
        Active_Material_ID := 0;
        Active_Bin_ID := 0;
        Excess_Alarm := FALSE;
        Status_Message := 'Auto [Step 7]: Settling Delay in progress...';
        Completion_Timer(IN := TRUE, PT := Effective_Delay);
        IF Completion_Timer.Q THEN
            Completion_Timer(IN := FALSE);
            Current_Step := 8;
        END_IF;

    8:
        Active_Material_ID := 0;
        Active_Bin_ID := 0;
        Excess_Alarm := FALSE;
        Sequence_Complete := TRUE;
        GVL.Auto_Sequence_Complete := TRUE;
        IF NOT GVL.Semi_Auto_Sequence_Complete THEN
            Status_Message := 'Auto [Step 8]: Auto Finished. Waiting for Semi-Auto to complete...';
        ELSE
            Status_Message := 'Auto [Step 8]: Cycle Sequences Complete';
        END_IF;
END_CASE;

(* Synchronize physical output arrays to GVL *)
FOR i := 1 TO 6 DO
    GVL.Auto_Bin[i] := Auto_Bin[i];
    GVL.auto_bin_cutoff[i] := auto_bin_cutoff[i];
    GVL.auto_bin_motor[i] := auto_bin_motor[i];
END_FOR;

(* Synchronize live cycle progress to outputs *)
Auto_Current_Batch_Cycle := GVL.Current_Batch_Cycle;
Auto_Completed_Batch_Cycles := GVL.Completed_Batch_Cycles;
Auto_All_Cycles_Complete := GVL.All_Cycles_Complete;

(* ---- FB_Samyak_Control.st ---- *)
(* ==========================================
   POU: FB_Samyak_Control
   ========================================== *)

=== DECLARATION ===
FUNCTION_BLOCK FB_Samyak_Control
VAR_INPUT
    Com_Slot      : BYTE := 1;     (* PLC COM port *)
    Slave_Dev_ID  : BYTE := 1;     (* Samyak slave ID *)
    iDivisor      : REAL := 10.0;  (* Scale factor: Weight_Scaled = Raw / iDivisor *)
    xTare_In      : BOOL;           (* Logic tare pulse *)
    xManual_Tare  : BOOL;           (* HMI/manual tare pulse *)
END_VAR

VAR_OUTPUT
    xStatus_Done   : BOOL;
    xStatus_Busy   : BOOL;
    xStatus_Error  : BOOL;
    iTotalErrCount : INT := 0;
    xLine_Fault    : BOOL;
    Weight_Raw     : DINT;
    Weight_Scaled  : REAL;
    wError_Code    : WORD; (* Check PLC & SAMYAK BaudRate, DevId, Parity; also check PLC serial port LED blink status and RS485 connection if error repeats *)
END_VAR

VAR
    fbRead         : ModRtuMast;
    fbTare         : ModRtuMast;
    iStep          : INT := 0;
    Samyak_Buffer  : ARRAY[0..17] OF WORD;
    wTareCommand   : WORD := 1;

    rtTareTrig     : R_TRIG;
    rtErrTrig      : R_TRIG;
    tStuckWatchdog : TON;
    tRecoveryTimer : TON;

    xTareReq       : BOOL := FALSE; (* Internal tare request latch *)
END_VAR

=== IMPLEMENTATION ===

(* --- 1) Error Tracking + Auto Recovery --- *)
tStuckWatchdog(IN := (fbRead.Busy OR fbTare.Busy), PT := T#2000MS);

rtErrTrig(CLK := (fbRead.Error OR fbTare.Error));
IF rtErrTrig.Q THEN
    iTotalErrCount := iTotalErrCount + 1;
END_IF

IF fbRead.Done OR fbTare.Done THEN
    iTotalErrCount := 0;
    xLine_Fault := FALSE;
END_IF

IF iTotalErrCount >= 10 THEN
    xLine_Fault := TRUE;
END_IF

tRecoveryTimer(IN := xLine_Fault, PT := T#5S);
IF tRecoveryTimer.Q THEN
    iTotalErrCount := 0;
    xLine_Fault := FALSE;
END_IF

IF tStuckWatchdog.Q THEN
    iStep := 99;
END_IF

(* Capture tare request from either input pulse *)
rtTareTrig(CLK := xTare_In OR xManual_Tare);
IF rtTareTrig.Q THEN
    xTareReq := TRUE;
END_IF

(* --- 2) Modbus State Machine --- *)
CASE iStep OF

    0:  (* Continuous Read *)
        fbTare(Execute := FALSE);

        fbRead(
            Execute := NOT (fbRead.Done OR fbRead.Error OR fbRead.Busy)
                       AND NOT xTareReq
                       AND NOT xLine_Fault,
            COM     := Com_Slot,
            Serv    := Slave_Dev_ID,
            FCT     := 3,
            Addr    := 0,
            Nb      := 2,
            Data    := ADR(Samyak_Buffer[0]),
            Timeout := 400,
            Done    => xStatus_Done,
            Busy    => xStatus_Busy,
            Error   => xStatus_Error,
            ErrorID => wError_Code
        );

        IF xStatus_Done THEN
            Weight_Raw := TO_DINT(SHL(TO_DWORD(Samyak_Buffer[1]), 16) OR TO_DWORD(Samyak_Buffer[0]));
            Weight_Scaled := TO_REAL(Weight_Raw) / iDivisor;
        END_IF

        IF xTareReq THEN
            iStep := 1;
        END_IF

    1:  (* Port Release *)
        fbRead(Execute := FALSE);
        IF NOT fbRead.Busy THEN
            iStep := 2;
        END_IF

    2:  (* Execute Tare *)
        fbTare(
            Execute := TRUE,
            COM     := Com_Slot,
            Serv    := Slave_Dev_ID,
            FCT     := 6,
            Addr    := 16,
            Nb      := 1,
            Data    := ADR(wTareCommand),
            Timeout := 1000,
            Done    => xStatus_Done,
            Busy    => xStatus_Busy,
            Error   => xStatus_Error,
            ErrorID => wError_Code
        );

        IF fbTare.Done OR fbTare.Error THEN
            xTareReq := FALSE;
            iStep := 3;
        END_IF

    3:  (* Return to Read *)
        fbTare(Execute := FALSE);
        IF NOT fbTare.Busy THEN
            iStep := 0;
        END_IF

    99: (* Emergency Recovery *)
        fbRead(Execute := FALSE);
        fbTare(Execute := FALSE);

        IF NOT (fbRead.Busy OR fbTare.Busy) THEN
            iTotalErrCount := 0;
            iStep := 0;
        END_IF

END_CASE

(* ---- FB_Samyak_Multi.st ---- *)
(* ==========================================
   POU: FB_Samyak_Multi
   ========================================== *)

=== DECLARATION ===
//SAMYAK 4016 Multi Slave Unit Customised Block
//Note: This FB_Samyak_Multi name is impotrtant when you create new POU.

FUNCTION_BLOCK FB_Samyak_Multi
VAR_INPUT
    Com_Slot      : BYTE := 1;    (* Port Number *)
    iSlaveCount   : INT := 1;     (* How many slaves active: 1 to 4 *)
    arrSlaveIDs   : ARRAY[1..4] OF BYTE := [1, 2, 3, 4]; (* Unit IDs *)
    arrDivisor    : ARRAY[1..4] OF REAL := [10.0, 10.0, 10.0, 10.0]; (* Scaling per Unit *)
    arrTare_In    : ARRAY[1..4] OF BOOL; (* Individual Tare triggers *)
END_VAR

VAR_OUTPUT
    arrWeight_Scaled : ARRAY[1..4] OF REAL; (* Scaled result per unit *)
    arrLine_Fault    : ARRAY[1..4] OF BOOL; (* Fault status per unit *)
    arrErrCount      : ARRAY[1..4] OF INT;  (* Error count per unit *)
    iCurrent_ID      : BYTE;                (* Current ID being polled *)
    xStatus_Busy     : BOOL;                (* Overall Bus Busy *)
END_VAR

VAR
    (* Internal ModRtuMast Instances *)
    fbRead         : ModRtuMast;
    fbTare         : ModRtuMast;

    (* Polling Control *)
    iStep          : INT := 0;
    iIdx           : INT := 1;    (* Current Loop Index *)
    Samyak_Buffer  : ARRAY[0..17] OF WORD;
    wTareCommand   : WORD := 1;

    (* Unique Timer/Trigger Instances *)
    rtTareTrig     : R_TRIG;
    rtErrTrig      : R_TRIG;
    tWatchdog      : TON;
    tRecovery      : TON;
END_VAR

=== IMPLEMENTATION ===

(* --- 1. INDIVIDUAL UNIT MONITORING --- *)
iCurrent_ID := arrSlaveIDs[iIdx];

(* Watchdog for Bus Hangs *)
tWatchdog(IN := (fbRead.Busy OR fbTare.Busy), PT := T#2000MS);
xStatus_Busy := fbRead.Busy OR fbTare.Busy;

(* Error Tracking for Current Index *)
rtErrTrig(CLK := (fbRead.Error OR fbTare.Error));
IF rtErrTrig.Q THEN
    arrErrCount[iIdx] := arrErrCount[iIdx] + 1;
END_IF

(* Reset on Success *)
IF fbRead.Done OR fbTare.Done THEN
    arrErrCount[iIdx] := 0;
    arrLine_Fault[iIdx] := FALSE;
END_IF

(* Line Fault Activation (10 errors) *)
IF arrErrCount[iIdx] >= 10 THEN
    arrLine_Fault[iIdx] := TRUE;
END_IF

(* Auto-Recovery pulse (5s) *)
tRecovery(IN := arrLine_Fault[iIdx], PT := T#5S);
IF tRecovery.Q THEN
    arrErrCount[iIdx] := 0;
    arrLine_Fault[iIdx] := FALSE;
END_IF

IF tWatchdog.Q THEN iStep := 99; END_IF

(* Check Tare for active slave *)
rtTareTrig(CLK := arrTare_In[iIdx]);

(* --- 2. SEQUENTIAL STATE MACHINE --- *)
CASE iStep OF

    0: (* READ CURRENT SLAVE *)
        fbTare(Execute := FALSE);
        fbRead(
            Execute := NOT (fbRead.Done OR fbRead.Error OR fbRead.Busy)
                       AND NOT rtTareTrig.Q AND NOT arrLine_Fault[iIdx],
            COM     := Com_Slot,
            Serv    := arrSlaveIDs[iIdx],
            FCT     := 3, Addr := 0, Nb := 2,
            Data    := ADR(Samyak_Buffer[0]), Timeout := 400
        );

        IF fbRead.Done THEN
            (* Scale weight using the array-based divisor for this specific index *)
            arrWeight_Scaled[iIdx] := TO_REAL(TO_DINT(SHL(TO_DWORD(Samyak_Buffer[1]), 16) OR TO_DWORD(Samyak_Buffer[0]))) / arrDivisor[iIdx];
            iStep := 10; (* Switch to next slave *)
        END_IF

        IF fbRead.Error THEN iStep := 10; END_IF (* Move on if error *)
        IF rtTareTrig.Q THEN iStep := 1; END_IF  (* Priority: Tare current unit *)

    1: (* PORT RELEASE *)
        fbRead(Execute := FALSE);
        IF NOT fbRead.Busy THEN iStep := 2; END_IF

    2: (* WRITE TARE FOR CURRENT SLAVE *)
        fbTare(
            Execute := TRUE,
            COM := Com_Slot, Serv := arrSlaveIDs[iIdx],
            FCT := 6, Addr := 16, Nb := 1,
            Data := ADR(wTareCommand), Timeout := 1000
        );

        IF fbTare.Done OR fbTare.Error THEN
            arrTare_In[iIdx] := FALSE; (* Reset manual trigger *)
            iStep := 3;
        END_IF

    3: (* CLEANUP *)
        fbTare(Execute := FALSE);
        IF NOT fbTare.Busy THEN iStep := 10; END_IF

    10: (* INDEX ROTATION *)
        iIdx := iIdx + 1;
        IF iIdx > iSlaveCount THEN
            iIdx := 1; (* Back to first slave *)
        END_IF
        iStep := 0;

    99: (* EMERGENCY RESET *)
        fbRead(Execute := FALSE); fbTare(Execute := FALSE);
        IF NOT (fbRead.Busy OR fbTare.Busy) THEN iStep := 0; END_IF

END_CASE

(* ---- sample_read_two_weights.st ---- *)
// ============================================================================
// FUNCTION BLOCK: sample_read_two_weights
// Method 3: Continuous Hardware Modbus Master Polling Table
// Replaces BLINK oscillator with a single ModRtuMast round-robin state machine.
// Automatically polls Auto Indicator (Node 1) and Semi-Auto Indicator (Node 2),
// scales raw DINT readings, and writes directly into GVL.load_cell_auto and
// GVL.load_cell_semi_auto with watchdog protection and communication diagnostics.
// ============================================================================

FUNCTION_BLOCK sample_read_two_weights
VAR_INPUT
    Enable               : BOOL := TRUE;       // Enable continuous cyclic polling
    Com_Slot             : BYTE := 1;          // PLC COM port number (e.g., COM1 = 1)
    Slave_Auto_ID        : BYTE := 1;          // Modbus Slave ID for Auto Scale Indicator
    Slave_Semi_ID        : BYTE := 2;          // Modbus Slave ID for Semi-Auto Scale Indicator
    iDivisor_Auto        : REAL := 10.0;       // Scale factor: Weight = Raw / Divisor
    iDivisor_Semi        : REAL := 10.0;       // Scale factor: Weight = Raw / Divisor
    Reg_Address          : WORD := 0;          // Starting register address for weight (Holding Reg)
    Reg_Quantity         : WORD := 2;          // Number of registers (2 words = 32-bit integer/float)
    Timeout_MS           : UINT := 400;        // Response timeout in milliseconds
    Gap_Time             : TIME := T#15MS;     // Inter-request line settling delay (RS485 turnaround)
END_VAR

VAR_OUTPUT
    Weight_Auto          : REAL;               // Scaled live weight for Auto scale -> GVL.load_cell_auto
    Weight_Semi          : REAL;               // Scaled live weight for Semi-Auto scale -> GVL.load_cell_semi_auto
    Weight_Raw_Auto      : DINT;               // Raw 32-bit value from Auto indicator
    Weight_Raw_Semi      : DINT;               // Raw 32-bit value from Semi-Auto indicator
    Auto_Scale_Online    : BOOL;               // Health flag: TRUE when Auto indicator is responding
    Semi_Scale_Online    : BOOL;               // Health flag: TRUE when Semi-Auto indicator is responding
    Current_Slave_Polled : BYTE;               // Currently active polled slave address
    Current_Slot_Index   : INT;                // 1 = Auto Indicator Slot, 2 = Semi-Auto Indicator Slot
    Poll_Cycles          : UDINT;              // Total completed round-robin polling cycles
    Total_Error_Count    : UDINT;              // Cumulative communication timeout/error count
    Status_Message       : STRING(80);         // Diagnostic status text for HMI
END_VAR

VAR
    fbModbus             : ModRtuMast;         // Single ModRtuMast instance for the entire bus
    iStep                : INT := 0;           // State machine: 0=Init, 1=Dispatch, 2=Wait, 3=Parse, 4=Gap
    iSlot                : INT := 1;           // 1 = Auto, 2 = Semi-Auto

    Buffer_Auto          : ARRAY[0..3] OF WORD;// Receive buffer for Auto indicator
    Buffer_Semi          : ARRAY[0..3] OF WORD;// Receive buffer for Semi-Auto indicator

    tWatchdog            : TON;                // Watchdog timer for bus protection
    tGapDelay            : TON;                // Inter-request gap delay timer

    xDone                : BOOL;
    xBusy                : BOOL;
    xError               : BOOL;
    wErrorCode           : ERROR_ID;
END_VAR

// ----------------------------------------------------------------------------
// Execution Body
// ----------------------------------------------------------------------------

IF NOT Enable THEN
    fbModbus(Execute := FALSE);
    iStep := 0;
    iSlot := 1;
    Status_Message := 'Polling Disabled';
    tGapDelay(IN := FALSE);
    tWatchdog(IN := FALSE);
    RETURN;
END_IF;

// 1. Driver Watchdog Protection
tWatchdog(IN := fbModbus.Busy, PT := T#2000MS);
IF tWatchdog.Q THEN
    iStep := 99; // Force emergency recovery if port locks
END_IF;

// 2. Round-Robin Master Polling Table State Machine
CASE iStep OF
    0: // Initialize Polling Table
        iSlot := 1;
        Current_Slot_Index := iSlot;
        Current_Slave_Polled := Slave_Auto_ID;
        fbModbus(Execute := FALSE);
        Status_Message := 'Modbus Master Polling Initialized';
        iStep := 1;

    1: // Dispatch Query for Current Slot
        Current_Slot_Index := iSlot;
        IF iSlot = 1 THEN
            Current_Slave_Polled := Slave_Auto_ID;
            fbModbus(
                Execute := TRUE,
                COM     := Com_Slot,
                Serv    := Slave_Auto_ID,
                FCT     := 3, // Read Holding Registers
                Addr    := Reg_Address,
                Nb      := Reg_Quantity,
                Data    := ADR(Buffer_Auto[0]),
                Timeout := Timeout_MS,
                Done    => xDone,
                Busy    => xBusy,
                Error   => xError,
                ErrorID => wErrorCode
            );
            Status_Message := CONCAT('Polling Auto Scale (Node ', CONCAT(BYTE_TO_STRING(Slave_Auto_ID), ')...'));
        ELSE
            Current_Slave_Polled := Slave_Semi_ID;
            fbModbus(
                Execute := TRUE,
                COM     := Com_Slot,
                Serv    := Slave_Semi_ID,
                FCT     := 3,
                Addr    := Reg_Address,
                Nb      := Reg_Quantity,
                Data    := ADR(Buffer_Semi[0]),
                Timeout := Timeout_MS,
                Done    => xDone,
                Busy    => xBusy,
                Error   => xError,
                ErrorID => wErrorCode
            );
            Status_Message := CONCAT('Polling Semi-Auto Scale (Node ', CONCAT(BYTE_TO_STRING(Slave_Semi_ID), ')...'));
        END_IF;
        iStep := 2;

    2: // Await Driver Response
        IF fbModbus.Done THEN
            fbModbus(Execute := FALSE);
            iStep := 3; // Advance to Parse Data
        ELSIF fbModbus.Error THEN
            fbModbus(Execute := FALSE);
            Total_Error_Count := Total_Error_Count + 1;
            IF iSlot = 1 THEN
                Auto_Scale_Online := FALSE;
                Status_Message := CONCAT('Auto Scale Comm Error ID: ', INT_TO_STRING(ERROR_ID_TO_INT(wErrorCode)));
            ELSE
                Semi_Scale_Online := FALSE;
                Status_Message := CONCAT('Semi-Auto Scale Comm Error ID: ', INT_TO_STRING(ERROR_ID_TO_INT(wErrorCode)));
            END_IF;
            iStep := 4; // Advance to Gap delay
        END_IF;

    3: // Parse Received Modbus Data into Scaled Weight
        IF iSlot = 1 THEN
            Weight_Raw_Auto := TO_DINT(SHL(TO_DWORD(Buffer_Auto[1]), 16) OR TO_DWORD(Buffer_Auto[0]));
            IF iDivisor_Auto <> 0.0 THEN
                Weight_Auto := TO_REAL(Weight_Raw_Auto) / iDivisor_Auto;
            ELSE
                Weight_Auto := TO_REAL(Weight_Raw_Auto);
            END_IF;
            GVL.load_cell_auto := Weight_Auto;
            Auto_Scale_Online := TRUE;
        ELSE
            Weight_Raw_Semi := TO_DINT(SHL(TO_DWORD(Buffer_Semi[1]), 16) OR TO_DWORD(Buffer_Semi[0]));
            IF iDivisor_Semi <> 0.0 THEN
                Weight_Semi := TO_REAL(Weight_Raw_Semi) / iDivisor_Semi;
            ELSE
                Weight_Semi := TO_REAL(Weight_Raw_Semi);
            END_IF;
            GVL.load_cell_semi_auto := Weight_Semi;
            Semi_Scale_Online := TRUE;
            Poll_Cycles := Poll_Cycles + 1;
        END_IF;
        iStep := 4;

    4: // Inter-Frame Line Gap Delay (Allows RS485 Transceivers to Settle)
        tGapDelay(IN := TRUE, PT := Gap_Time);
        IF tGapDelay.Q THEN
            tGapDelay(IN := FALSE);
            // Alternate Table Slot: 1 -> 2 -> 1 -> 2 ...
            IF iSlot = 1 THEN
                iSlot := 2;
            ELSE
                iSlot := 1;
            END_IF;
            iStep := 1; // Dispatch next query
        END_IF;

    99: // Emergency Driver Reset / Bus Recovery
        fbModbus(Execute := FALSE);
        tGapDelay(IN := FALSE);
        IF NOT fbModbus.Busy THEN
            iStep := 0;
        END_IF;
END_CASE;

(* ---- Semi_Auto_Batching_V14.st ---- *)
FUNCTION_BLOCK Semi_Auto_Batching_V14
VAR_INPUT
    Start_Button : BOOL;                                 // Command pulse/signal to start or resume the semi-auto batching sequence
    E_Stop_Active : BOOL;                                // Emergency Stop circuit status (NC contact: TRUE = Healthy/Run permitted, FALSE = E-Stop tripped)
    Reset : BOOL;                                        // System reset pulse (clears active steps, outputs, alarms, and error flags)
    Semi_Auto_Bin_Material_Mapping : ARRAY[1..10] OF INT;// Array mapping physical Silos 1..10 to Recipe Material IDs (1..20, 0 = Silo skipped)
    Semi_Auto_Coarse_To_Fine_Speed : ARRAY[1..10] OF REAL;// Weight offset threshold (kg) before target to transition from Coarse to Fine feeding
    Semi_Auto_Bin_Tolerance : ARRAY[1..10] OF REAL;      // Allowable weight tolerance window (±kg) around target weight for each silo
    Inter_Bin_Delay : TIME;                              // Settling delay duration after completing a bin before advancing to the next
    Excess_Allowed : BOOL;                               // Overfill handling policy: TRUE = proceed if target is exceeded, FALSE = raise alarm and halt
    load_cell_value : REAL;                              // Live gross weight input reading from the Semi-Auto scale load cell (kg)
    Target_Batch_Cycles : INT;                           // Target number of batch cycle repetitions configured from HMI (defaults to 1)
    Next_Cycle_Start : BOOL;                             // Command pulse/signal to start next batch cycle after hoppers are emptied
    Empty_Weight_Limit : REAL;                           // Maximum scale weight limit (kg) for scales to qualify as empty before starting next cycle
END_VAR
VAR_OUTPUT
    Semi_Auto_Bin : ARRAY[1..10] OF BOOL;                // Coarse feeding valve / gate actuation command outputs for Silos 1..10
    semi_auto_bin_cutoff : ARRAY[1..10] OF BOOL;         // Fine feeding valve / vibrator cutoff actuation command outputs for Silos 1..10
    semi_auto_bin_motor : ARRAY[1..10] OF BOOL;          // Feeder / screw conveyor motor run commands for Silos 1..10
    Actual_Weights : ARRAY[1..10] OF REAL;               // Net material weight (kg) successfully dosed for each silo in the current cycle
    Sequence_Complete : BOOL;                            // Handshake flag: TRUE when all mapped Semi-Auto silos have completed dosing and settling
    Active_Material_ID : INT;                            // Recipe Material ID currently being dosed (1..20, 0 when idle/complete)
    Active_Bin_ID : INT;                                 // Physical Silo index currently being dosed (1..10, 0 when idle/complete)
    Active_Target_Weight : REAL;                         // Target weight setpoint (kg) of the ingredient currently being dosed
    Active_Live_Weight : REAL;                           // Live net/tared weight (kg) accumulated into the scale for the active silo
    Current_Step : INT;                                  // Real-time sequence step:
                                                         //   0   = Idle / Waiting for Start
                                                         //   1..10 = Dosing Silos 1..10 (feeding coarse/fine)
                                                         //   31  = Settling delay in progress
                                                         //   32  = Sequence complete
    Cycle_Manager_State : INT;                           // Master supervisory cycle manager state:
                                                         //   0   = System Idle / Stopped
                                                         //   1   = Running active batch cycle
                                                         //   4   = All target batch cycles completed successfully
                                                         //   5   = Paused between cycles (Cycle Hold active)
    Excess_Alarm : BOOL;                                 // Overfill alarm: TRUE when dosed weight exceeds target + tolerance (with Excess_Allowed=FALSE)
    Error_Code : INT;                                    // Fault diagnostic code:
                                                         //   0   = No Error / System Healthy
                                                         //   1   = Duplicate Material ID mapped across Auto and Semi-Auto
                                                         //   2   = Material index out of range (must be 1..20)
                                                         //   3   = Recipe weight is less than (Coarse_To_Fine_Speed + Tolerance)
                                                         //   4   = Initial scale tare error (scale not empty before start)
                                                         //   21  = Scale overload protection triggered (> 500 kg)
    Semi_Auto_Current_Batch_Cycle : INT;                 // Active batch cycle number currently processing (1..Target_Batch_Cycles)
    Semi_Auto_Completed_Batch_Cycles : INT;              // Total number of batch cycle loops completed successfully
    Semi_Auto_All_Cycles_Complete : BOOL;                // Master flag: TRUE when all Target_Batch_Cycles have finished
    Status_Message : STRING(80);                         // Real-time human-readable process status and diagnostic text message
END_VAR
VAR
    bin_last_weight : REAL;
    actual_bin : REAL;
    target_weight : REAL;
    cutoff_trigger_weight : REAL;
    min_tol_weight : REAL;
    max_tol_weight : REAL;
    Paused_By_EStop : BOOL;
    Effective_Delay : TIME;
    Mat_Idx : INT;
    i : INT;
    Last_Batch_Cycle : INT;
    Transition_Timer : TON;
    Completion_Timer : TON;
    Simulation_Mode : BOOL;
    Sim_Rate : REAL;
    Sim_Timer : TON;
    Start_Sim_Weight : REAL;
    Discharge_Active : BOOL;
    Run_Last : BOOL;
    Run_Rising : BOOL;
END_VAR

(* Semi-Auto Batching FB V14 with Full Diagnostics, Step Tracking, and Precise Status Reporting *)

Effective_Delay := Inter_Bin_Delay;
IF Effective_Delay = T#0S THEN
    Effective_Delay := T#2S;
END_IF;

(* Track Master Cycle State *)
IF Target_Batch_Cycles > 0 THEN
    GVL.Target_Batch_Cycles := Target_Batch_Cycles;
END_IF;

(* Master Cycle State & Start Synchronization *)
Run_Rising := GVL.Run AND NOT Run_Last;
Run_Last := GVL.Run;

IF GVL.Run THEN
    IF Sequence_Complete AND GVL.Auto_Sequence_Complete THEN
        IF GVL.Current_Batch_Cycle >= GVL.Target_Batch_Cycles AND GVL.Target_Batch_Cycles > 0 THEN
            Cycle_Manager_State := 4;
        ELSE
            Cycle_Manager_State := 5;
        END_IF;
    ELSE
        Cycle_Manager_State := 1;
    END_IF;
ELSE
    Cycle_Manager_State := 0;
    Current_Step := 0;
    Last_Batch_Cycle := 0;
    Sequence_Complete := FALSE;
    GVL.Semi_Auto_Sequence_Complete := FALSE;
END_IF;

(* On fresh batch start (rising edge of Run), ensure clean start from Step 0 *)
IF Run_Rising THEN
    Current_Step := 0;
    Last_Batch_Cycle := 0;
    Sequence_Complete := FALSE;
    GVL.Semi_Auto_Sequence_Complete := FALSE;
END_IF;

(* 1. SEMI-AUTO RECIPE TOTALS & ACTIVE SILO COUNT *)
GVL.Semi_Auto_Total_Target_Weight := 0.0;
GVL.Semi_Auto_Material_Count := 0;
FOR i := 1 TO 10 DO
    IF Semi_Auto_Bin_Material_Mapping[i] > 0 AND Semi_Auto_Bin_Material_Mapping[i] <= 20 THEN
        IF GVL.Recipe_Weights[Semi_Auto_Bin_Material_Mapping[i]] > 0.0 THEN
            GVL.Semi_Auto_Total_Target_Weight := GVL.Semi_Auto_Total_Target_Weight + GVL.Recipe_Weights[Semi_Auto_Bin_Material_Mapping[i]];
            GVL.Semi_Auto_Material_Count := GVL.Semi_Auto_Material_Count + 1;
        END_IF;
    END_IF;
END_FOR;

(* 2. HARD RESET INTERLOCK *)
IF Reset OR GVL.Reset THEN
    FOR i := 1 TO 10 DO
        Semi_Auto_Bin[i] := FALSE;
        semi_auto_bin_cutoff[i] := FALSE;
        semi_auto_bin_motor[i] := FALSE;
        Actual_Weights[i] := 0.0;
        GVL.Semi_Auto_Bin[i] := FALSE;
        GVL.semi_auto_bin_cutoff[i] := FALSE;
        GVL.semi_auto_bin_motor[i] := FALSE;
        GVL.Semi_Auto_Weights[i] := 0.0;
    END_FOR;
    Sequence_Complete := FALSE;
    GVL.Semi_Auto_Sequence_Complete := FALSE;
    Active_Material_ID := 0;
    Active_Bin_ID := 0;
    Active_Target_Weight := 0.0;
    Active_Live_Weight := 0.0;
    GVL.Semi_Auto_Active_Target_Weight := 0.0;
    GVL.Semi_Auto_Active_Live_Weight := 0.0;
    GVL.Semi_Auto_Active_Mat := 0;
    GVL.Semi_Auto_Active_Bin := 0;
    GVL.Semi_Auto_Excess_Alarm := FALSE;
    Excess_Alarm := FALSE;
    Error_Code := 0;
    Paused_By_EStop := FALSE;
    Current_Step := 0;
    Last_Batch_Cycle := 0;
    Cycle_Manager_State := 0;
    Semi_Auto_Current_Batch_Cycle := 0;
    Semi_Auto_Completed_Batch_Cycles := 0;
    Semi_Auto_All_Cycles_Complete := FALSE;
    bin_last_weight := 0.0;
    Start_Sim_Weight := 0.0;
    Run_Last := FALSE;
    Run_Rising := FALSE;
    Transition_Timer(IN := FALSE);
    Completion_Timer(IN := FALSE);
    Sim_Timer(IN := FALSE);
    Status_Message := 'Semi-Auto [Reset]: System Reset Complete - System Idle';

    (* Clean Auto-Clearing: Reset has been processed by both blocks *)
    GVL.Reset := FALSE;
    RETURN;
END_IF;

(* 3. E-STOP PAUSE / HOLD LOGIC (NC Contact: FALSE = Pressed/Tripped, TRUE = Healthy) *)
IF NOT E_Stop_Active OR NOT GVL.E_Stop_Active THEN
    Paused_By_EStop := TRUE;
END_IF;

IF Paused_By_EStop THEN
    FOR i := 1 TO 10 DO
        Semi_Auto_Bin[i] := FALSE;
        semi_auto_bin_cutoff[i] := FALSE;
        semi_auto_bin_motor[i] := FALSE;
    END_FOR;
    IF NOT E_Stop_Active OR NOT GVL.E_Stop_Active THEN
        Status_Message := CONCAT('Semi-Auto [PAUSED]: E-Stop Active at Step ', INT_TO_STRING(Current_Step));
    ELSE
        Status_Message := CONCAT('Semi-Auto [HOLD]: E-Stop Cleared. Press Start to Resume Step ', INT_TO_STRING(Current_Step));
        IF Start_Button OR GVL.Start_Button THEN
            Paused_By_EStop := FALSE;
        END_IF;
    END_IF;
    Sim_Timer(IN := FALSE);
    Transition_Timer(IN := FALSE);
    Completion_Timer(IN := FALSE);
    RETURN;
END_IF;

(* 4. CYCLE COMPLETE / HOLD STATE *)
IF Cycle_Manager_State = 5 THEN
    Status_Message := 'Semi-Auto [Cycle Complete]: Waiting for scale empty & Next_Cycle_Start...';
END_IF;

(* 5. SEQUENCE START (FOR CYCLE 1 AND REPEAT CYCLES) *)
IF GVL.Run AND Cycle_Manager_State <> 5 THEN
    IF Current_Step = 0 THEN
        (* Initial cycle start *)
        Last_Batch_Cycle := GVL.Current_Batch_Cycle;
        Current_Step := 1;
        bin_last_weight := load_cell_value;
        Sequence_Complete := FALSE;
        GVL.Semi_Auto_Sequence_Complete := FALSE;
        Excess_Alarm := FALSE;
        Error_Code := 0;
        FOR i := 1 TO 10 DO
            Actual_Weights[i] := 0.0;
            Semi_Auto_Bin[i] := FALSE;
            semi_auto_bin_cutoff[i] := FALSE;
            semi_auto_bin_motor[i] := FALSE;
        END_FOR;
    ELSIF Current_Step = 32 AND GVL.Current_Batch_Cycle <> Last_Batch_Cycle THEN
        (* Advance to next cycle loop (Cycle 2, 3, etc.) *)
        Last_Batch_Cycle := GVL.Current_Batch_Cycle;
        Current_Step := 1;
        bin_last_weight := load_cell_value;
        Sequence_Complete := FALSE;
        GVL.Semi_Auto_Sequence_Complete := FALSE;
        Excess_Alarm := FALSE;
        Error_Code := 0;
        FOR i := 1 TO 10 DO
            Actual_Weights[i] := 0.0;
            Semi_Auto_Bin[i] := FALSE;
            semi_auto_bin_cutoff[i] := FALSE;
            semi_auto_bin_motor[i] := FALSE;
        END_FOR;
    END_IF;
END_IF;

CASE Current_Step OF
    0:
        Active_Material_ID := 0;
        Active_Bin_ID := 0;
        Excess_Alarm := FALSE;
        Sequence_Complete := FALSE;
        FOR i := 1 TO 10 DO
            Semi_Auto_Bin[i] := FALSE;
            semi_auto_bin_cutoff[i] := FALSE;
            semi_auto_bin_motor[i] := FALSE;
        END_FOR;
        Active_Target_Weight := GVL.Semi_Auto_Active_Target_Weight;
        Active_Live_Weight := 0.0;
        IF Error_Code = 0 AND Cycle_Manager_State <> 5 THEN
            Status_Message := 'Semi-Auto [Step 0 - Idle]: Ready - Waiting for Run Signal';
        END_IF;

    1..10:
        (* Skip any bin where Material Mapping is 0, > 20, or Recipe Weight is 0 *)
        WHILE Current_Step >= 1 AND Current_Step <= 10 DO
            Mat_Idx := Semi_Auto_Bin_Material_Mapping[Current_Step];
            IF Mat_Idx = 0 OR Mat_Idx > 20 OR GVL.Recipe_Weights[Mat_Idx] <= 0.0 THEN
                Semi_Auto_Bin[Current_Step] := FALSE;
                semi_auto_bin_cutoff[Current_Step] := FALSE;
                semi_auto_bin_motor[Current_Step] := FALSE;
                Actual_Weights[Current_Step] := 0.0;
                IF Current_Step = 10 THEN
                    Current_Step := 31;
                    EXIT;
                ELSE
                    Current_Step := Current_Step + 1;
                END_IF;
            ELSE
                EXIT; (* Valid active recipe silo found *)
            END_IF;
        END_WHILE;

        IF Current_Step = 31 THEN
            Active_Material_ID := 0;
            Active_Bin_ID := 0;
            Active_Target_Weight := 0.0;
            Active_Live_Weight := 0.0;
            GVL.Semi_Auto_Active_Target_Weight := 0.0;
            GVL.Semi_Auto_Active_Live_Weight := 0.0;
            Status_Message := 'Semi-Auto [Step 31]: Settling Delay in progress...';
            Completion_Timer(IN := TRUE, PT := Effective_Delay);
            IF Completion_Timer.Q THEN
                Completion_Timer(IN := FALSE);
                Current_Step := 32;
            END_IF;
        ELSE
            Mat_Idx := Semi_Auto_Bin_Material_Mapping[Current_Step];
            target_weight := GVL.Recipe_Weights[Mat_Idx];

            Active_Target_Weight := target_weight;
            GVL.Semi_Auto_Active_Target_Weight := target_weight;

            cutoff_trigger_weight := target_weight - Semi_Auto_Coarse_To_Fine_Speed[Current_Step];
            min_tol_weight := target_weight - Semi_Auto_Bin_Tolerance[Current_Step];
            max_tol_weight := target_weight + Semi_Auto_Bin_Tolerance[Current_Step];

            actual_bin := load_cell_value - bin_last_weight;
            IF actual_bin < 0.0 THEN
                actual_bin := 0.0;
            END_IF;
            Actual_Weights[Current_Step] := actual_bin;
            Active_Live_Weight := actual_bin;
            GVL.Semi_Auto_Active_Live_Weight := actual_bin;
            Active_Material_ID := Mat_Idx;
            Active_Bin_ID := Current_Step;

            IF load_cell_value > 500.0 THEN
                Error_Code := 21;
                GVL.Error_Code := 21;
                Status_Message := CONCAT('Semi-Auto [Step ', CONCAT(INT_TO_STRING(Current_Step), ']: STUCK - Error 21: Scale Overloaded (> 500 kg)!'));
                Sequence_Complete := TRUE;
                GVL.Semi_Auto_Sequence_Complete := TRUE;
                Paused_By_EStop := TRUE;
            END_IF;

            IF actual_bin < cutoff_trigger_weight THEN
                Semi_Auto_Bin[Current_Step] := TRUE;
                semi_auto_bin_cutoff[Current_Step] := FALSE;
                semi_auto_bin_motor[Current_Step] := TRUE;
                Excess_Alarm := FALSE;
                Status_Message := CONCAT('Semi-Auto [Step ', CONCAT(INT_TO_STRING(Current_Step), ']: Coarse Feeding'));
            ELSIF actual_bin < min_tol_weight THEN
                Semi_Auto_Bin[Current_Step] := FALSE;
                semi_auto_bin_cutoff[Current_Step] := TRUE;
                semi_auto_bin_motor[Current_Step] := TRUE;
                Excess_Alarm := FALSE;
                Status_Message := CONCAT('Semi-Auto [Step ', CONCAT(INT_TO_STRING(Current_Step), ']: Fine Feeding'));
            ELSIF actual_bin > max_tol_weight THEN
                Semi_Auto_Bin[Current_Step] := FALSE;
                semi_auto_bin_cutoff[Current_Step] := FALSE;
                semi_auto_bin_motor[Current_Step] := FALSE;
                IF Excess_Allowed THEN
                    Excess_Alarm := FALSE;
                    Status_Message := CONCAT('Semi-Auto [Step ', CONCAT(INT_TO_STRING(Current_Step), ']: Excess Allowed - Advancing'));
                    bin_last_weight := load_cell_value;
                    Active_Target_Weight := 0.0;
                    Active_Live_Weight := 0.0;
                    GVL.Semi_Auto_Active_Target_Weight := 0.0;
                    GVL.Semi_Auto_Active_Live_Weight := 0.0;
                    IF Current_Step = 10 THEN
                        Current_Step := 31;
                    ELSE
                        Current_Step := Current_Step + 1;
                    END_IF;
                ELSE
                    Excess_Alarm := TRUE;
                    Status_Message := CONCAT('Semi-Auto [Step ', CONCAT(INT_TO_STRING(Current_Step), ']: STUCK - Excess Weight! Reduce weight or enable Excess Allowed.'));
                END_IF;
            ELSE
                Semi_Auto_Bin[Current_Step] := FALSE;
                semi_auto_bin_cutoff[Current_Step] := FALSE;
                semi_auto_bin_motor[Current_Step] := FALSE;
                Excess_Alarm := FALSE;
                bin_last_weight := load_cell_value;
                Active_Target_Weight := 0.0;
                Active_Live_Weight := 0.0;
                GVL.Semi_Auto_Active_Target_Weight := 0.0;
                GVL.Semi_Auto_Active_Live_Weight := 0.0;
                Status_Message := CONCAT('Semi-Auto [Step ', CONCAT(INT_TO_STRING(Current_Step), ']: Target Reached - Advancing'));
                IF Current_Step = 10 THEN
                    Current_Step := 31;
                ELSE
                    Current_Step := Current_Step + 1;
                END_IF;
            END_IF;
        END_IF;

    31:
        Active_Material_ID := 0;
        Active_Bin_ID := 0;
        Excess_Alarm := FALSE;
        Status_Message := 'Semi-Auto [Step 31]: Settling Delay in progress...';
        Completion_Timer(IN := TRUE, PT := Effective_Delay);
        IF Completion_Timer.Q THEN
            Completion_Timer(IN := FALSE);
            Current_Step := 32;
        END_IF;

    32:
        Active_Material_ID := 0;
        Active_Bin_ID := 0;
        Excess_Alarm := FALSE;
        Sequence_Complete := TRUE;
        GVL.Semi_Auto_Sequence_Complete := TRUE;
        IF NOT GVL.Auto_Sequence_Complete THEN
            Status_Message := 'Semi-Auto [Step 32]: Semi-Auto Finished. Waiting for Auto to complete...';
        ELSE
            Status_Message := 'Semi-Auto [Step 32]: Cycle Sequences Complete';
        END_IF;
END_CASE;

(* Synchronize physical output arrays to GVL *)
FOR i := 1 TO 10 DO
    GVL.Semi_Auto_Bin[i] := Semi_Auto_Bin[i];
    GVL.semi_auto_bin_cutoff[i] := semi_auto_bin_cutoff[i];
    GVL.semi_auto_bin_motor[i] := semi_auto_bin_motor[i];
END_FOR;

(* Synchronize live cycle progress to outputs *)
Semi_Auto_Current_Batch_Cycle := GVL.Current_Batch_Cycle;
Semi_Auto_Completed_Batch_Cycles := GVL.Completed_Batch_Cycles;
Semi_Auto_All_Cycles_Complete := GVL.All_Cycles_Complete;

(* ---- batching13.st ---- *)
PROGRAM batching13
VAR
    Auto_Ctrl : Auto_Batching_V13;
    Semi_Auto_Ctrl : Semi_Auto_Batching_V13;

    (* Sub-Block Diagnostic Indicators *)
    Auto_Err : INT;
    Auto_Msg : STRING;

    Semi_Auto_Err : INT;
    Semi_Auto_Msg : STRING;

    Auto_Complete : BOOL;
    Semi_Auto_Complete : BOOL;

    (* Repetitive Cycle Status *)
    Completed_Batch_Cycles : INT;      // Total completed batch cycle loops
    All_Cycles_Complete : BOOL;         // Indicator for full set completion

    (* Diagnostics & Interlocks *)
    Status_Message : STRING;

    i : INT;
    j : INT;
    Duplicate_Found : BOOL;
    Invalid_Material_Range : BOOL;
    Weight_Limit_Error : BOOL;

    (* Cycle Manager state variables *)
    Cycle_Manager_State : INT;         // State index for loop management
    Internal_FB_Start : BOOL;          // Controlled command to restart sub-blocks
END_VAR

(* 1. STARTUP CONFIGURATION, RECIPE TOTALS, AND WEIGHT CHECKS *)
Duplicate_Found := FALSE;
Invalid_Material_Range := FALSE;
Weight_Limit_Error := FALSE;

(* Calculate Auto Total Target Weight & Material Count *)
GVL.Auto_Total_Target_Weight := 0.0;
GVL.Auto_Material_Count := 0;
FOR i := 1 TO 6 DO
    (* Check 2: Out of Range (Auto) *)
    IF GVL.Auto_Bin_Material_Mapping[i] < 0 OR GVL.Auto_Bin_Material_Mapping[i] > 20 THEN
        Invalid_Material_Range := TRUE;
    END_IF;

    (* Check 1: Duplicate Cross-Array Material ID *)
    IF GVL.Auto_Bin_Material_Mapping[i] <> 0 AND GVL.Auto_Bin_Material_Mapping[i] <= 20 THEN
        FOR j := 1 TO 10 DO
            IF GVL.Auto_Bin_Material_Mapping[i] = GVL.Semi_Auto_Bin_Material_Mapping[j] THEN
                Duplicate_Found := TRUE;
            END_IF;
        END_FOR;
    END_IF;

    (* Accumulate Auto Total Target Weight and Active Count *)
    IF GVL.Auto_Bin_Material_Mapping[i] > 0 AND GVL.Auto_Bin_Material_Mapping[i] <= 20 THEN
        IF GVL.Recipe_Weights[GVL.Auto_Bin_Material_Mapping[i]] > 0.0 THEN
            GVL.Auto_Total_Target_Weight := GVL.Auto_Total_Target_Weight + GVL.Recipe_Weights[GVL.Auto_Bin_Material_Mapping[i]];
            GVL.Auto_Material_Count := GVL.Auto_Material_Count + 1;

            (* Check 3: Recipe weight is less than Cutoff + Tolerance *)
            IF GVL.Recipe_Weights[GVL.Auto_Bin_Material_Mapping[i]] < (GVL.Auto_Coarse_To_Fine_speed[i] + GVL.Auto_Bin_Tolerance[i]) THEN
                Weight_Limit_Error := TRUE;
            END_IF;
        END_IF;
    END_IF;
END_FOR;

(* Calculate Semi-Auto Total Target Weight & Material Count *)
GVL.Semi_Auto_Total_Target_Weight := 0.0;
GVL.Semi_Auto_Material_Count := 0;
FOR j := 1 TO 10 DO
    (* Check 2: Out of Range (Semi-Auto) *)
    IF GVL.Semi_Auto_Bin_Material_Mapping[j] < 0 OR GVL.Semi_Auto_Bin_Material_Mapping[j] > 20 THEN
        Invalid_Material_Range := TRUE;
    END_IF;

    (* Accumulate Semi-Auto Total Target Weight and Active Count *)
    IF GVL.Semi_Auto_Bin_Material_Mapping[j] > 0 AND GVL.Semi_Auto_Bin_Material_Mapping[j] <= 20 THEN
        IF GVL.Recipe_Weights[GVL.Semi_Auto_Bin_Material_Mapping[j]] > 0.0 THEN
            GVL.Semi_Auto_Total_Target_Weight := GVL.Semi_Auto_Total_Target_Weight + GVL.Recipe_Weights[GVL.Semi_Auto_Bin_Material_Mapping[j]];
            GVL.Semi_Auto_Material_Count := GVL.Semi_Auto_Material_Count + 1;

            (* Check 3: Recipe weight check (Semi-Auto) *)
            IF GVL.Recipe_Weights[GVL.Semi_Auto_Bin_Material_Mapping[j]] < (GVL.Semi_Auto_Coarse_To_Fine_speed[j] + GVL.Semi_Auto_Bin_Tolerance[j]) THEN
                Weight_Limit_Error := TRUE;
            END_IF;
        END_IF;
    END_IF;
END_FOR;

(* Configuration Error Resolution *)
IF Duplicate_Found THEN
    GVL.Error_Code := 1;
    Status_Message := 'Error 1: Duplicate Material ID mapped in Auto and Semi-Auto!';
ELSIF Invalid_Material_Range THEN
    GVL.Error_Code := 2;
    Status_Message := 'Error 2: Material Index configuration out of range (1..20)!';
ELSIF Weight_Limit_Error THEN
    GVL.Error_Code := 3;
    Status_Message := 'Error 3: Recipe weight is less than Cutoff + Tolerance!';
ELSE
    IF GVL.Error_Code <= 3 THEN
        GVL.Error_Code := 0;
    END_IF;
END_IF;

(* Abort / Hard Reset Interlock *)
IF (GVL.Error_Code >= 1 AND GVL.Error_Code <= 3) OR GVL.Reset THEN
    FOR i := 1 TO 6 DO
        GVL.Auto_Bin[i] := FALSE;
        GVL.auto_bin_cutoff[i] := FALSE;
        GVL.auto_bin_motor[i] := FALSE;
        GVL.Auto_Weights[i] := 0.0;
    END_FOR;

    FOR i := 1 TO 10 DO
        GVL.Semi_Auto_Bin[i] := FALSE;
        GVL.semi_auto_bin_cutoff[i] := FALSE;
        GVL.semi_auto_bin_motor[i] := FALSE;
        GVL.Semi_Auto_Weights[i] := 0.0;
    END_FOR;

    Internal_FB_Start := FALSE;
    Auto_Ctrl(Start_Button := FALSE, E_Stop_Active := FALSE, Reset := GVL.Reset, load_cell_value := GVL.load_cell_auto, Inter_Bin_Delay := GVL.Auto_Inter_Bin_Delay, Excess_Allowed := GVL.Auto_Excess_Allowed);
    Semi_Auto_Ctrl(Start_Button := FALSE, E_Stop_Active := FALSE, Reset := GVL.Reset, load_cell_value := GVL.load_cell_semi_auto, Inter_Bin_Delay := GVL.Semi_Auto_Inter_Bin_Delay, Excess_Allowed := GVL.Semi_Auto_Excess_Allowed);

    GVL.Auto_Active_Target_Weight := 0.0;
    GVL.Auto_Active_Live_Weight := 0.0;
    GVL.Semi_Auto_Active_Target_Weight := 0.0;
    GVL.Semi_Auto_Active_Live_Weight := 0.0;

    Auto_Complete := TRUE;
    Semi_Auto_Complete := TRUE;
    All_Cycles_Complete := TRUE;

    GVL.Cycle_Hold_Active := FALSE;
    GVL.Run := FALSE;
    Cycle_Manager_State := 0;

    IF GVL.Reset THEN
        GVL.Error_Code := 0;
        GVL.Current_Batch_Cycle := 0;
        GVL.Target_Batch_Cycles := 0;
        GVL.Start_Button := FALSE;
        Completed_Batch_Cycles := 0;
        Status_Message := 'System Reset Activated';
        Auto_Complete := FALSE;
        Semi_Auto_Complete := FALSE;
        All_Cycles_Complete := FALSE;

        GVL.Auto_Active_Mat := 0;
        GVL.Auto_Active_Bin := 0;
        GVL.Semi_Auto_Active_Mat := 0;
        GVL.Semi_Auto_Active_Bin := 0;
        GVL.Auto_Excess_Alarm := FALSE;
        GVL.Semi_Auto_Excess_Alarm := FALSE;

        (* Auto-clearing trigger: set Reset back to FALSE *)
        GVL.Reset := FALSE;
    END_IF;
    RETURN;
END_IF;

(* 2. REPETITIVE CYCLE MANAGER STATE MACHINE WITH PRE-RUN INITIAL TOLERANCE CHECK *)
CASE Cycle_Manager_State OF
    0: (* IDLE STATE *)
        Internal_FB_Start := FALSE;
        All_Cycles_Complete := FALSE;
        GVL.Cycle_Hold_Active := FALSE;
        GVL.Run := FALSE;
        IF GVL.Error_Code = 0 AND Status_Message <> 'Error: Target Batch Cycles is 0!' AND Status_Message <> 'Error 4: Scale weight exceeds Initial Tolerance!' THEN
            Status_Message := 'System Ready';
        END_IF;

        IF GVL.Start_Button THEN
            (* Guard 1: Target_Batch_Cycles must be > 0 *)
            IF GVL.Target_Batch_Cycles <= 0 THEN
                GVL.Run := FALSE;
                Status_Message := 'Error: Target Batch Cycles is 0!';
            (* Guard 2: Check Initial Tolerance ONLY before setting Run = TRUE *)
            ELSIF (GVL.load_cell_auto > GVL.Auto_Initial_Tolerance OR GVL.load_cell_auto < (-GVL.Auto_Initial_Tolerance)) OR
                  (GVL.load_cell_semi_auto > GVL.Semi_Auto_Initial_Tolerance OR GVL.load_cell_semi_auto < (-GVL.Semi_Auto_Initial_Tolerance)) THEN
                GVL.Run := FALSE;
                GVL.Error_Code := 4;
                Status_Message := 'Error 4: Scale weight exceeds Initial Tolerance!';
            ELSE
                GVL.Error_Code := 0;
                GVL.Current_Batch_Cycle := 1;
                Completed_Batch_Cycles := 0;

                Auto_Complete := FALSE;
                Semi_Auto_Complete := FALSE;

                GVL.Run := TRUE;
                Cycle_Manager_State := 1;
            END_IF;
        END_IF;

    1: (* RUN STATE (Run Sub-Blocks - Initial Tolerance is NOT checked here while pouring) *)
        Internal_FB_Start := TRUE;
        GVL.Run := TRUE;
        Status_Message := CONCAT('Running Batch Cycle ', INT_TO_STRING(GVL.Current_Batch_Cycle));

        (* Monitor completion of active step *)
        IF Auto_Complete AND Semi_Auto_Complete THEN
            Cycle_Manager_State := 2;
        END_IF;

    2: (* CHECK REPEAT CYCLE STATE *)
        Completed_Batch_Cycles := GVL.Current_Batch_Cycle;
        GVL.Run := TRUE;

        (* Block cycle repeat in case of active error *)
        IF GVL.Current_Batch_Cycle < GVL.Target_Batch_Cycles AND GVL.Error_Code = 0 THEN
            (* Hold cycle loop progression *)
            GVL.Cycle_Hold_Active := TRUE;
            Internal_FB_Start := FALSE; (* Reset FBs to 0 while waiting in hold *)
            Cycle_Manager_State := 5; // Go to hold wait state
        ELSE
            (* All loop cycles complete *)
            Cycle_Manager_State := 4;
        END_IF;

    5: (* PAUSED BETWEEN CYCLES *)
        Internal_FB_Start := FALSE; (* Keeps sub-blocks in Step 0 *)
        GVL.Run := TRUE;
        Status_Message := CONCAT('Cycle ', CONCAT(INT_TO_STRING(GVL.Current_Batch_Cycle), ' Complete. Empty scale to 0 and release Cycle Hold.'));

        IF NOT GVL.Cycle_Hold_Active THEN
            (* Check Initial Tolerance before starting next cycle *)
            IF (GVL.load_cell_auto > GVL.Auto_Initial_Tolerance OR GVL.load_cell_auto < (-GVL.Auto_Initial_Tolerance)) OR
               (GVL.load_cell_semi_auto > GVL.Semi_Auto_Initial_Tolerance OR GVL.load_cell_semi_auto < (-GVL.Semi_Auto_Initial_Tolerance)) THEN
                GVL.Run := FALSE;
                GVL.Error_Code := 4;
                Status_Message := 'Error 4: Scale weight exceeds Initial Tolerance!';
                GVL.Cycle_Hold_Active := TRUE; (* Keep hold active until scale is emptied *)
            ELSE
                GVL.Error_Code := 0;
                GVL.Current_Batch_Cycle := GVL.Current_Batch_Cycle + 1;
                Auto_Complete := FALSE;
                Semi_Auto_Complete := FALSE;
                Cycle_Manager_State := 1; (* Start next cycle! *)
            END_IF;
        END_IF;

    4: (* SEQUENCE FULLY COMPLETED STATE *)
        Internal_FB_Start := FALSE;
        All_Cycles_Complete := TRUE;
        GVL.Run := FALSE;
        GVL.Start_Button := FALSE; (* Auto-turn off Start_Button when process completes! *)
        Status_Message := 'All Batch Cycles Completed';

        Cycle_Manager_State := 0;
END_CASE;

(* 3. CONCURRENT EXECUTION OF FB INSTANCES WITH GVL ARRAYS & LIVE ACTIVE WEIGHTS *)
Auto_Ctrl(
    Start_Button := Internal_FB_Start,
    E_Stop_Active := GVL.E_Stop_Active,
    Reset := GVL.Reset,
    load_cell_value := GVL.load_cell_auto,
    Auto_Bin_Material_Mapping := GVL.Auto_Bin_Material_Mapping,
    Auto_Coarse_To_Fine_speed := GVL.Auto_Coarse_To_Fine_speed,
    Auto_Bin_Tolerance := GVL.Auto_Bin_Tolerance,
    Inter_Bin_Delay := GVL.Auto_Inter_Bin_Delay,
    Excess_Allowed := GVL.Auto_Excess_Allowed,
    Auto_Bin => GVL.Auto_Bin,
    auto_bin_cutoff => GVL.auto_bin_cutoff,
    auto_bin_motor => GVL.auto_bin_motor,
    Actual_Weights => GVL.Auto_Weights,
    Sequence_Complete => Auto_Complete,
    Active_Material_ID => GVL.Auto_Active_Mat,
    Active_Bin_ID => GVL.Auto_Active_Bin,
    Active_Target_Weight => GVL.Auto_Active_Target_Weight,
    Active_Live_Weight => GVL.Auto_Active_Live_Weight,
    Excess_Alarm => GVL.Auto_Excess_Alarm,
    Error_Code => Auto_Err,
    Status_Message => Auto_Msg
);

Semi_Auto_Ctrl(
    Start_Button := Internal_FB_Start,
    E_Stop_Active := GVL.E_Stop_Active,
    Reset := GVL.Reset,
    load_cell_value := GVL.load_cell_semi_auto,
    Semi_Auto_Bin_Material_Mapping := GVL.Semi_Auto_Bin_Material_Mapping,
    Semi_Auto_Coarse_To_Fine_speed := GVL.Semi_Auto_Coarse_To_Fine_speed,
    Semi_Auto_Bin_Tolerance := GVL.Semi_Auto_Bin_Tolerance,
    Inter_Bin_Delay := GVL.Semi_Auto_Inter_Bin_Delay,
    Excess_Allowed := GVL.Semi_Auto_Excess_Allowed,
    Semi_Auto_Bin => GVL.Semi_Auto_Bin,
    semi_auto_bin_cutoff => GVL.semi_auto_bin_cutoff,
    semi_auto_bin_motor => GVL.semi_auto_bin_motor,
    Actual_Weights => GVL.Semi_Auto_Weights,
    Sequence_Complete => Semi_Auto_Complete,
    Active_Material_ID => GVL.Semi_Auto_Active_Mat,
    Active_Bin_ID => GVL.Semi_Auto_Active_Bin,
    Active_Target_Weight => GVL.Semi_Auto_Active_Target_Weight,
    Active_Live_Weight => GVL.Semi_Auto_Active_Live_Weight,
    Excess_Alarm => GVL.Semi_Auto_Excess_Alarm,
    Error_Code => Semi_Auto_Err,
    Status_Message => Semi_Auto_Msg
);

(* Runtime Error Mapping & Aggregation *)
IF Auto_Err <> 0 THEN
    GVL.Error_Code := Auto_Err;
    Status_Message := CONCAT('Auto Error: ', Auto_Msg);
    Auto_Complete := TRUE;
    Semi_Auto_Complete := TRUE;
    All_Cycles_Complete := TRUE;
    GVL.Run := FALSE;
    GVL.Start_Button := FALSE;
ELSIF Semi_Auto_Err <> 0 THEN
    GVL.Error_Code := Semi_Auto_Err;
    Status_Message := CONCAT('Semi-Auto Error: ', Semi_Auto_Msg);
    Auto_Complete := TRUE;
    Semi_Auto_Complete := TRUE;
    All_Cycles_Complete := TRUE;
    GVL.Run := FALSE;
    GVL.Start_Button := FALSE;
ELSIF Cycle_Manager_State = 0 AND GVL.Error_Code <= 3 THEN
    GVL.Error_Code := 0;
END_IF;

(* ---- batching14.st ---- *)
(* ==========================================
   POU: batching14
   ========================================== *)

=== DECLARATION ===
PROGRAM batching14
VAR
	Auto_Ctrl: Auto_Batching_V14;
	Semi_Auto_Ctrl: Semi_Auto_Batching_V14;
	Auto_Complete: BOOL;
	Semi_Auto_Complete: BOOL;
	Auto_Err: INT;
	Auto_Msg: STRING;
	Semi_Auto_Err: INT;
	Semi_Auto_Msg: STRING;
	FB_Samyak_Multi_1: FB_Samyak_Multi;
	arrSlaveIDs: ARRAY[1..4] OF BYTE := [1, 2, 0, 0];
	arrDivisor: ARRAY[1..4] OF REAL := [10.0, 10.0, 1.0, 1.0];
	arrTare_In: ARRAY[1..4] OF BOOL;
	Weight_Scaled_Array: ARRAY[1..4] OF REAL;
	arrLine_Fault: ARRAY[1..4] OF BOOL;
END_VAR
